# B&R Automation Studio project CombinedLinenSoiledA9KAN (part 16)

#### hlDFIICyclic.st - Cyclic code
```iecst
(********************************************************************
 * COPYRIGHT -- Microsoft
 ********************************************************************
 * Program: hlDFII
 * File: hlDFIICyclic.st
 * Author: hunholz
 * Created: April 05, 2011
 * Changed: November 14, 2011
 ********************************************************************
 * Implementation of program hlDFII
 ********************************************************************)

PROGRAM _CYCLIC

	// Init
	IF IFmnParam.Out.xParamOK AND NOT _xInitDone THEN

		brwcsconv(ADR(_sMNo), ADR(IFmnParam.Out.utfMachineNumber), 1);

		_xInitDone := TRUE;

	END_IF

	IF NOT _xReady AND IFmnEth.Out.xDataValid AND IFmnParam.Out.xParamOK AND HLDFII_RUN_CLIENT THEN

		//**********************
		// INITIALISIERUNG
		//***********************

		_sDBserv := USINT_TO_STRING(IFmnEth.Out.IP.bNetId1);
		_sDBserv := CONCAT(_sDBserv,'.');
		_sOkt := USINT_TO_STRING(IFmnEth.Out.IP.bNetId2);
		_sDBserv := CONCAT(_sDBserv,_sOkt);
		_sDBserv := CONCAT(_sDBserv,'.');
		_sOkt := USINT_TO_STRING(IFmnEth.Out.IP.bNetId3+hlDFIIPar.Mac.bDBservReg);
		_sDBserv := CONCAT(_sDBserv,_sOkt);
		_sDBserv := CONCAT(_sDBserv,'.');
		_sOkt := USINT_TO_STRING(hlDFIIPar.Mac.bDBservAdr);
		_sDBserv := CONCAT(_sDBserv,_sOkt);

		_sUdpHost := _sDBserv;

		brsstrcpy(ADR(_sInstance),ADR(hlDFIIPar.Mac.sServInst));

		IF hlDFIIPar.Mac.wDBservPort <> 0 THEN

			// Wenn der Port <> 0 ist, wird der SQL-Server direkt über den Port angesprochen

			_sDBserv := CONCAT(_sDBserv, ':');
			_sOkt 	 := UINT_TO_STRING(hlDFIIPar.Mac.wDBservPort);
			_sDBserv := CONCAT(_sDBserv, _sOkt);

		ELSE

			// Wenn mit der Instanz gearbeitet wird, muss auf dem PC der SQL-Browser-Dienst laufen

			IF LEN(_sInstance) > 0 THEN

				REPEAT

					_iFound := FIND(_sInstance,' ');

					IF _iFound <> 0 THEN
						_sInstance := DELETE(_sInstance,1,_iFound);
					END_IF

					UNTIL
					_iFound = 0 OR LEN(_sInstance) = 0
				END_REPEAT

				IF LEN(_sInstance) > 0 THEN
					_sDBserv := CONCAT(_sDBserv, '\');
					_sDBserv := CONCAT(_sDBserv, _sInstance);
				END_IF

			END_IF

		END_IF

		_xReady := TRUE;

		// UDP-Log vorbereiten

		_UdpOpen.enable	 := TRUE;
		_UdpOpen.pIfAddr := 0;
		_UdpOpen.port	 := HLDFII_UDP_PORT_LOG4NET;
		_UdpOpen.options := udpOPT_BROADCAST;

	ELSIF _xReady THEN

		//***********************************
		// ZYKLISCHE ABARBEITUNG
		//***********************************

		hlDFIIStat.wStatus := 0;

		//*********************************************************************************
		// Request scheduler
		//*********************************************************************************

		IF _eCmdStep = eCMD_SQLREQ_IDLE THEN

			CASE _wCmdCnt OF

				0:
					// Uhrzeit holen
					IF _bEventGetTime = 1 THEN
						// Auftrag starten
						_eCmdStep := eCMD_SQLREQ_WRITE_GETTIME;
						_bEventGetTime := 2;
					END_IF
				1:
					// Maschine registrieren
					IF _bEventRegMach = 1 AND brwcscmp(ADR(IFmnParam.Out.utfMachineNumber),ADR(MNPARAM_INVALID_MACHINENO)) <> 0 THEN
						// Auftrag starten
						_eCmdStep := eCMD_SQLREQ_WRITE_REGMACH;
						_bEventRegMach := 2;
					END_IF

				2:
					IF _xWaitReqProgByCatIsZero THEN

						IF IFhlDFII.In.ReqProgByCat.wRequest = 0 THEN

							_xWaitReqProgByCatIsZero := FALSE;
							IFhlDFII.Out.RespProgByCat.wResponse := 0;

						END_IF

					ELSE

						// Prüfen ob eine Programmnummer gelesen werden soll
						IF IFhlDFII.In.ReqProgByCat.wRequest = 1 OR IFhlDFII.In.ReqProgByCat.wRequest = 2 THEN

							IF IFhlDFII.Out.xConnected THEN

								_xWaitReqProgByCatIsZero := TRUE;
								// Auftrag starten
								_eCmdStep := eCMD_SQLREQ_GET_PROG_BY_CAT;
								IFhlDFII.Out.RespProgByCat.wResponse := ERR_FUB_BUSY;

							ELSE

								_xWaitReqProgByCatIsZero := TRUE;
								IFhlDFII.Out.RespProgByCat.wResponse := HLDFII_STAT_NO_CONNECTION;

							END_IF

						END_IF

					END_IF

				3:
					IF _xWaitReqMsgEvtIsZero THEN

						IF IFhlDFII.In.ReqMsgEvt.wRequest = 0 THEN
							_xWaitReqMsgEvtIsZero := FALSE;
							IFhlDFII.Out.RespMsgEvt.wResponse := 0;
						END_IF

					ELSE

						IF IFhlDFII.Out.xConnected THEN

							// Prüfen ob Meldungsevents geschrieben werden sollen
							IF IFhlDFII.In.ReqMsgEvt.wRequest = 1 THEN

								_xWaitReqMsgEvtIsZero := TRUE;

								IF IFhlDFII.In.ReqMsgEvt.bCntLines > 0 THEN
									_eCmdStep := eCMD_SQLREQ_WRITE_MSG;
									IFhlDFII.Out.RespMsgEvt.wResponse := ERR_FUB_BUSY;
								ELSE
									IFhlDFII.Out.RespMsgEvt.wResponse := IFhlDFII.In.ReqMsgEvt.wRequest;
								END_IF

							END_IF

						ELSE

							_xWaitReqMsgEvtIsZero := TRUE;
							IFhlDFII.Out.RespMsgEvt.wResponse := HLDFII_STAT_NO_CONNECTION;

						END_IF

					END_IF

				4:
					IF _xWaitReqCntBatchIsZero THEN

						IF IFhlDFII.In.ReqCntBatchEvt.wRequest = 0 THEN

							_xWaitReqCntBatchIsZero := FALSE;
							IFhlDFII.Out.RespCntBatchEvt.wResponse := 0;

						END_IF

					ELSE

						IF IFhlDFII.Out.xConnected THEN

							// Prüfen ob Zähler-Posten-Events geschrieben werden sollen
							IF IFhlDFII.In.ReqCntBatchEvt.wRequest = 1 THEN

								_xWaitReqCntBatchIsZero := TRUE;

								IF IFhlDFII.In.ReqCntBatchEvt.bCntLines > 0 THEN
									_eCmdStep := eCMD_SQLREQ_WRITE_CNTBATCHEVT;
									IFhlDFII.Out.RespCntBatchEvt.wResponse := ERR_FUB_BUSY;
								ELSE
									IFhlDFII.Out.RespCntBatchEvt.wResponse  := IFhlDFII.In.ReqCntBatchEvt.wRequest;
								END_IF
							END_IF

						ELSE

							_xWaitReqCntBatchIsZero := TRUE;
							IFhlDFII.Out.RespCntBatchEvt.wResponse := HLDFII_STAT_NO_CONNECTION;

						END_IF

					END_IF
				5:
					IF _xWaitReqCntCntIsZero THEN

						IF IFhlDFII.In.ReqCntCntEvt.wRequest = 0 THEN

							_xWaitReqCntCntIsZero := FALSE;
							IFhlDFII.Out.RespCntCntEvt.wResponse := 0;

						END_IF

					ELSE

						IF IFhlDFII.Out.xConnected THEN

							// Prüfen ob Zähler-Zähler-Events geschrieben werden sollen
							IF IFhlDFII.In.ReqCntCntEvt.wRequest = 1 THEN

								_xWaitReqCntCntIsZero := TRUE;

								IF IFhlDFII.In.ReqCntCntEvt.bCntLines > 0 THEN
									_eCmdStep := eCMD_SQLREQ_WRITE_CNTCNTEVT;
									IFhlDFII.Out.RespCntCntEvt.wResponse := ERR_FUB_BUSY;
								ELSE
									IFhlDFII.Out.RespCntCntEvt.wResponse  := IFhlDFII.In.ReqCntCntEvt.wRequest;
								END_IF
							END_IF

						ELSE

							_xWaitReqCntCntIsZero := TRUE;
							IFhlDFII.Out.RespCntCntEvt.wResponse := HLDFII_STAT_NO_CONNECTION;

						END_IF

					END_IF
				6:
					IF _xWaitReqCntTimIsZero THEN

						IF IFhlDFII.In.ReqCntTimEvt.wRequest = 0 THEN

							_xWaitReqCntTimIsZero := FALSE;
							IFhlDFII.Out.RespCntTimEvt.wResponse := 0;

						END_IF

					ELSE

						IF IFhlDFII.Out.xConnected THEN

							// Prüfen ob Zähler-Zeit-Events geschrieben werden sollen
							IF IFhlDFII.In.ReqCntTimEvt.wRequest = 1 THEN

								_xWaitReqCntTimIsZero := TRUE;

								IF IFhlDFII.In.ReqCntTimEvt.bCntLines > 0 THEN
									_eCmdStep := eCMD_SQLREQ_WRITE_CNTTIMEVT;
									IFhlDFII.Out.RespCntTimEvt.wResponse := ERR_FUB_BUSY;
								ELSE
									IFhlDFII.Out.RespCntTimEvt.wResponse  := IFhlDFII.In.ReqCntTimEvt.wRequest;
								END_IF
							END_IF

						ELSE

							_xWaitReqCntTimIsZero := TRUE;
							IFhlDFII.Out.RespCntTimEvt.wResponse := HLDFII_STAT_NO_CONNECTION;

						END_IF

					END_IF
				7:
					IF _xWaitReqCntDosIsZero THEN

						IF IFhlDFII.In.ReqCntDosEvt.wRequest = 0 THEN

							_xWaitReqCntDosIsZero := FALSE;
							IFhlDFII.Out.RespCntDosEvt.wResponse := 0;

						END_IF

					ELSE

						IF IFhlDFII.Out.xConnected THEN

							// Prüfen ob Zähler-Dosier-Events geschrieben werden sollen
							IF IFhlDFII.In.ReqCntDosEvt.wRequest = 1 THEN

								_xWaitReqCntDosIsZero := TRUE;

								IF IFhlDFII.In.ReqCntDosEvt.bCntLines > 0 THEN
									_eCmdStep := eCMD_SQLREQ_WRITE_CNTDOSEVT;
									IFhlDFII.Out.RespCntDosEvt.wResponse := ERR_FUB_BUSY;
								ELSE
									IFhlDFII.Out.RespCntDosEvt.wResponse  := IFhlDFII.In.ReqCntDosEvt.wRequest;
								END_IF

							END_IF

						ELSE

							_xWaitReqCntDosIsZero := TRUE;
							IFhlDFII.Out.RespCntDosEvt.wResponse := HLDFII_STAT_NO_CONNECTION;

						END_IF

					END_IF

			END_CASE

		END_IF

		//*********************************************************************************
		// Aufträge ausführen
		//*********************************************************************************

		CASE _eCmdStep OF

			eCMD_SQLREQ_IDLE:

				IF TRUE THEN

					IF _bEventGetTime <> 3 THEN
						_wCmdCnt := 0;
					ELSIF _bEventRegMach <> 3 THEN
						_wCmdCnt := 1;
					ELSE
						_wHelpCmdCnt := (_wHelpCmdCnt + 1) MOD 6;
						_wCmdCnt := _wHelpCmdCnt + 2;
					END_IF

				ELSE

					_xReady := FALSE;

				END_IF

			//*****************************************************
			// Auftrag: Programm nach Kategorie auslesen
			//*****************************************************
			eCMD_SQLREQ_GET_PROG_BY_CAT:

				IF _eStep = eSQLREQ_STEP_WAITFORCOMMAND THEN
					IFhlDFII.Out.RespProgByCat.bProgramNo 		:= 0;
					IFhlDFII.Out.RespProgByCat.sProgramName 	:= '';
					IFhlDFII.Out.RespProgByCat.rSoilfactor 		:= 1.0;
					IFhlDFII.Out.RespProgByCat.wLoadrate 		:= 100;
					IFhlDFII.Out.RespProgByCat.wColorIdxFor 	:= 0;
					IFhlDFII.Out.RespProgByCat.wColorIdxBack 	:= 15;
					_eStep := eSQLREQ_STEP_GPBC;
					_eCmdStep := eCMD_SQLREQ_GET_PROG_BY_CAT_w;

				ELSIF _eStep = eSQLREQ_STEP_ERROR THEN

					IFhlDFII.Out.RespProgByCat.wResponse := HLDFII_MSG_PROGBYCAT_ERR;
					_eCmdStep := eCMD_SQLREQ_IDLE;

				END_IF

			eCMD_SQLREQ_GET_PROG_BY_CAT_w:

				IF _eStep = eSQLREQ_STEP_WAITFORCOMMAND THEN
					IFhlDFII.Out.RespProgByCat.wResponse := IFhlDFII.In.ReqProgByCat.wRequest;
					_eCmdStep := eCMD_SQLREQ_IDLE;
				ELSIF _eStep = eSQLREQ_STEP_ERROR THEN
					IFhlDFII.Out.RespProgByCat.wResponse := HLDFII_MSG_PROGBYCAT_ERR;
					_eCmdStep := eCMD_SQLREQ_IDLE;
				END_IF

			//*****************************************************
			// Meldungen schreiben
			//*****************************************************
			eCMD_SQLREQ_WRITE_MSG:

				IF _eStep = eSQLREQ_STEP_WAITFORCOMMAND THEN
					_bCntWrMsg := 1;
					_eStep := eSQLREQ_STEP_WRMSG;
					_eCmdStep := eCMD_SQLREQ_WRITE_MSG_w;
				ELSIF _eStep = eSQLREQ_STEP_ERROR THEN
					IFhlDFII.Out.RespMsgEvt.wResponse := HLDFII_MSG_MSGEVT_ERR;
					_eCmdStep := eCMD_SQLREQ_IDLE;
				END_IF

			eCMD_SQLREQ_WRITE_MSG_w:

				IF _eStep = eSQLREQ_STEP_WAITFORCOMMAND THEN
					IFhlDFII.Out.RespMsgEvt.wResponse := IFhlDFII.In.ReqMsgEvt.wRequest;
					_eCmdStep := eCMD_SQLREQ_IDLE;
				ELSIF _eStep = eSQLREQ_STEP_ERROR THEN
					IFhlDFII.Out.RespMsgEvt.wResponse := HLDFII_MSG_MSGEVT_ERR;
					_eCmdStep := eCMD_SQLREQ_IDLE;
				END_IF

			//*****************************************************
			// Posten-Zählevents schreiben
			//*****************************************************
			eCMD_SQLREQ_WRITE_CNTBATCHEVT:

				IF _eStep = eSQLREQ_STEP_WAITFORCOMMAND THEN
					_bCntWrCntBatchEvt := 1;
					_eStep := eSQLREQ_STEP_WRCNTBATCHEVT;
					_eCmdStep := eCMD_SQLREQ_WRITE_CNTBATCHEVT_w;
				ELSIF _eStep = eSQLREQ_STEP_ERROR THEN
					IFhlDFII.Out.RespCntBatchEvt.wResponse := HLDFII_MSG_CNTBATCHEVT_ERR;
					_eCmdStep := eCMD_SQLREQ_IDLE;
				END_IF

			eCMD_SQLREQ_WRITE_CNTBATCHEVT_w:

				IF _eStep = eSQLREQ_STEP_WAITFORCOMMAND THEN
					IFhlDFII.Out.RespCntBatchEvt.wResponse := IFhlDFII.In.ReqCntBatchEvt.wRequest;
					_eCmdStep := eCMD_SQLREQ_IDLE;
				ELSIF _eStep = eSQLREQ_STEP_ERROR THEN
					IFhlDFII.Out.RespCntBatchEvt.wResponse := HLDFII_MSG_CNTBATCHEVT_ERR;
					_eCmdStep := eCMD_SQLREQ_IDLE;
				END_IF

			//*****************************************************
			// Zählerevents schreiben
			//*****************************************************
			eCMD_SQLREQ_WRITE_CNTCNTEVT:

				IF _eStep = eSQLREQ_STEP_WAITFORCOMMAND THEN
					_bCntWrCntCntEvt := 1;
					_eStep := eSQLREQ_STEP_WRCNTCNTEVT;
					_eCmdStep := eCMD_SQLREQ_WRITE_CNTCNTEVT_w;
				ELSIF _eStep = eSQLREQ_STEP_ERROR THEN
					IFhlDFII.Out.RespCntCntEvt.wResponse := HLDFII_MSG_CNTCNTEVT_ERR;
					_eCmdStep := eCMD_SQLREQ_IDLE;
				END_IF

			eCMD_SQLREQ_WRITE_CNTCNTEVT_w:

				IF _eStep = eSQLREQ_STEP_WAITFORCOMMAND THEN
					IFhlDFII.Out.RespCntCntEvt.wResponse := IFhlDFII.In.ReqCntCntEvt.wRequest;
					_eCmdStep := eCMD_SQLREQ_IDLE;
				ELSIF _eStep = eSQLREQ_STEP_ERROR THEN
					IFhlDFII.Out.RespCntCntEvt.wResponse := HLDFII_MSG_CNTCNTEVT_ERR;
					_eCmdStep := eCMD_SQLREQ_IDLE;
				END_IF

			//*****************************************************
			// Zeitevents schreiben
			//*****************************************************
			eCMD_SQLREQ_WRITE_CNTTIMEVT:

				IF _eStep = eSQLREQ_STEP_WAITFORCOMMAND THEN
					_bCntWrCntTimeEvt := 1;
					_eStep := eSQLREQ_STEP_WRCNTTIMEVT;
					_eCmdStep := eCMD_SQLREQ_WRITE_CNTTIMEVT_w;
				ELSIF _eStep = eSQLREQ_STEP_ERROR THEN
					IFhlDFII.Out.RespCntTimEvt.wResponse := HLDFII_MSG_CNTTIMEVT_ERR;
					_eCmdStep := eCMD_SQLREQ_IDLE;
				END_IF

			eCMD_SQLREQ_WRITE_CNTTIMEVT_w:

				IF _eStep = eSQLREQ_STEP_WAITFORCOMMAND THEN
					IFhlDFII.Out.RespCntTimEvt.wResponse := IFhlDFII.In.ReqCntTimEvt.wRequest;
					_eCmdStep := eCMD_SQLREQ_IDLE;
				ELSIF _eStep = eSQLREQ_STEP_ERROR THEN
					IFhlDFII.Out.RespCntTimEvt.wResponse := HLDFII_MSG_CNTTIMEVT_ERR;
					_eCmdStep := eCMD_SQLREQ_IDLE;
				END_IF

			//*****************************************************
			// Dosierevents schreiben
			//*****************************************************
			eCMD_SQLREQ_WRITE_CNTDOSEVT:

				IF _eStep = eSQLREQ_STEP_WAITFORCOMMAND THEN
					_bCntWrCntDoseEvt := 1;
					_eStep := eSQLREQ_STEP_WRCNTDOSEVT;
					_eCmdStep := eCMD_SQLREQ_WRITE_CNTDOSEVT_W;
				ELSIF _eStep = eSQLREQ_STEP_ERROR THEN
					IFhlDFII.Out.RespCntDosEvt.wResponse := HLDFII_MSG_CNTDOSEVT_ERR;
					_eCmdStep := eCMD_SQLREQ_IDLE;
				END_IF

			eCMD_SQLREQ_WRITE_CNTDOSEVT_W:

				IF _eStep = eSQLREQ_STEP_WAITFORCOMMAND THEN
					IFhlDFII.Out.RespCntDosEvt.wResponse := IFhlDFII.In.ReqCntDosEvt.wRequest;
					_eCmdStep := eCMD_SQLREQ_IDLE;
				ELSIF _eStep = eSQLREQ_STEP_ERROR THEN
					IFhlDFII.Out.RespCntDosEvt.wResponse := HLDFII_MSG_CNTDOSEVT_ERR;
					_eCmdStep := eCMD_SQLREQ_IDLE;
				END_IF

			//*****************************************************
			// Maschine registrieren
			//*****************************************************
			eCMD_SQLREQ_WRITE_REGMACH:

				IF _eStep = eSQLREQ_STEP_WAITFORCOMMAND THEN
					_eStep := eSQLREQ_STEP_REGMACH;
					_eCmdStep := eCMD_SQLREQ_WRITE_REGMACH_w;
				ELSIF _eStep = eSQLREQ_STEP_ERROR THEN
					_bEventRegMach := 255;
					_eCmdStep := eCMD_SQLREQ_IDLE;
				END_IF

			eCMD_SQLREQ_WRITE_REGMACH_w:

				IF _eStep = eSQLREQ_STEP_WAITFORCOMMAND THEN
					_bEventRegMach := 3;
					_eCmdStep := eCMD_SQLREQ_IDLE;
				ELSIF _eStep = eSQLREQ_STEP_ERROR THEN
					_bEventRegMach := 255;
					_eCmdStep := eCMD_SQLREQ_IDLE;
				END_IF

			//*****************************************************
			// Uhrzeit vom DB-Server holen
			//*****************************************************
			eCMD_SQLREQ_WRITE_GETTIME:

				IF _eStep = eSQLREQ_STEP_WAITFORCOMMAND THEN
					_eStep := eSQLREQ_STEP_GETTIME;
					_eCmdStep := eCMD_SQLREQ_WRITE_GETTIME_w;
				ELSIF _eStep = eSQLREQ_STEP_ERROR THEN
					_bEventGetTime := 255;
					_eCmdStep := eCMD_SQLREQ_IDLE;
				END_IF

			eCMD_SQLREQ_WRITE_GETTIME_w:

				IF _eStep = eSQLREQ_STEP_WAITFORCOMMAND THEN
					_bEventGetTime := 3;
					_eCmdStep := eCMD_SQLREQ_IDLE;
				ELSIF _eStep = eSQLREQ_STEP_ERROR THEN
					_bEventGetTime := 255;
					_eCmdStep := eCMD_SQLREQ_IDLE;
				END_IF

		END_CASE

		//*********************************************************************************
		// Verbindung nach ablauf der Idletime abbauen, wenn keine Aktion ist
		//*********************************************************************************

		IF _eStep = eSQLREQ_STEP_ERROR THEN

			_eStep := eSQLREQ_STEP_DISCONNECT;

		ELSIF (_eCmdStep = eCMD_SQLREQ_IDLE) AND(_eStep = eSQLREQ_STEP_WAITFORCOMMAND) THEN

			_GTCurrent(enable := TRUE);

			IF _GTCurrent.DT1 > _GTlastAction.DT1 THEN

				IF DiffDT(_GTCurrent.DT1, _GTlastAction.DT1) > hlDFIIPar.Mac.wIdletimeDisconnect THEN

					// Idletime abgelaufen, Verbindung abbauen
					_eStep := eSQLREQ_STEP_DISCONNECT;

				END_IF

			END_IF

		ELSE

			_GTlastAction(enable := TRUE);

		END_IF

		//*********************************************************************************
		// Verbindung bei Bedarf aufbauen
		//*********************************************************************************

		IF _eCmdStep <> eCMD_SQLREQ_IDLE AND _eStep = eSQLREQ_STEP_STOP THEN

			_eStep := eSQLREQ_STEP_CONNECT;

		END_IF

		//*********************************************************************************
		// SQL-Befehle ausführen
		//*********************************************************************************

		CASE _eStep OF

			eSQLREQ_STEP_STOP:

			eSQLREQ_STEP_WAITFORCOMMAND:

			(* Verbinde Datenbank *)
			eSQLREQ_STEP_CONNECT:

				_DFII_Connect.enable := TRUE;
				_DFII_Connect.databaseSystem := DB_SYSTEM_MS_SQL;
				_DFII_Connect.pUserName := ADR('plc');
				_DFII_Connect.pPassword := ADR('plc');
				_DFII_Connect.pServerName := ADR(_sDBserv);
				_DFII_Connect.pDatabaseName := ADR(hlDFIIPar.Mac.sDBname);
				_eStep := eSQLREQ_STEP_CONNECT_r;

			(* Warte bis mit Datenbank verbunden *)
			eSQLREQ_STEP_CONNECT_r:

				_DFII_Connect();

				IF _DFII_Connect.status = ERR_OK THEN

					// Verbindung Erfolgreich

					IF _DFII_Connect.connectionIdent = 0 THEN

						// Wenn Verbindung nicht möglich, immer erst wieder Zeit holen und Maschine registrieren
						_bEventRegMach := 1;
						_bEventGetTime := 1;
						IFhlDFII.Out.xConnected := FALSE;

						// Fehler ist Clientseitig
						_sLogEntryI := 'Client Fault: Connect failed! ';
						_sLogEntryI := CONCAT(_sLogEntryI,_sDBserv);
						_eStep := eSQLREQ_STEP_LOGRB_ERROR;

					ELSE

						IFhlDFII.Out.xConnected := TRUE;

						_sLogEntryI := WSTRING_TO_STRING(IFmnParam.Out.utfMachineNumber);
						_sLogEntryI := CONCAT(_sLogEntryI, '-hlDFII$tSUCC$tCONNECT');
						_InsertRB(wPtrWrite := _wPtrRBwrite, wPtrRead := _wPtrRBread, wPtrStart := _wPtrRBstart);

						_lConnectionIdent := _DFII_Connect.connectionIdent;
						_eStep := eSQLREQ_STEP_WAITFORCOMMAND;
					END_IF

				ELSIF _DFII_Connect.status <> ERR_FUB_BUSY THEN

					// Wenn Verbindung nicht möglich, immer erst wieder Zeit holen und Maschine registrieren
					_bEventRegMach := 1;
					_bEventGetTime := 1;
					IFhlDFII.Out.xConnected := FALSE;

					// Verbindung fehlerbehaftet
					IF _DFII_Connect.connectionIdent <> 0 THEN

						// Fehler ist Serverseitig, Fehlermeldung holen

						_lConnectionIdent := _DFII_Connect.connectionIdent;
						_sAction := 'Connect failed:';
						_eStep := eSQLREQ_STEP_GET_ERROR;

					ELSE

						// Keine Verbindung zustande gekommen
						_sLogEntryI := 'Connect failed! ';
						_sLogEntryI := CONCAT(_sLogEntryI,_sDBserv);

						_eStep := eSQLREQ_STEP_LOGRB_ERROR;

					END_IF

				END_IF

			(* Baue Datenbankverbindung ab *)
			eSQLREQ_STEP_DISCONNECT:

				IF _lConnectionIdent <> 0 THEN
					_DFII_Disconnect.enable := TRUE;
					_DFII_Disconnect.connectionIdent := _lConnectionIdent;
					_eStep := eSQLREQ_STEP_DISCONNECT_r;
				ELSE
					_eStep := eSQLREQ_STEP_STOP;
				END_IF

			(* Warte bis Verbindung abgebaut ist *)
			eSQLREQ_STEP_DISCONNECT_r:

				_DFII_Disconnect();

				IF _DFII_Disconnect.status <> ERR_FUB_BUSY THEN

					// Verbindung erfolgreich unterbrochen

					_sLogEntryI := WSTRING_TO_STRING(IFmnParam.Out.utfMachineNumber);
					_sLogEntryI := CONCAT(_sLogEntryI, '-hlDFII$tSUCC$tDISCONNECT');
					_InsertRB(wPtrWrite := _wPtrRBwrite, wPtrRead := _wPtrRBread, wPtrStart := _wPtrRBstart);

					_eStep := eSQLREQ_STEP_STOP;
					_lConnectionIdent := 0;

				END_IF

			(* Lese Programmnummer aus Datenbank *)
			eSQLREQ_STEP_GPBC:

				_sCat := IFhlDFII.In.ReqProgByCat.sCategoryNo_In;

				brsstrcpy(ADR(_sSQLstring), ADR('SELECT [ProgramNo], [ProgramName], [CategoryName], [LoadFactor], [SoiledFactor], [fgColorIndex], [bgColorIndex]  FROM [dbo].[vwCatToProg01] WHERE [MachineID] = N$''));
				brsstrcat(ADR(_sSQLstring), ADR(_sMNo));
				IF (IFhlDFII.In.ReqProgByCat.wRequest = 2) THEN
					brsstrcat(ADR(_sSQLstring),ADR('$' AND  LTRIM(RTRIM(CategoryNoAlpha)) =  LTRIM(RTRIM($''));
				ELSE
					brsstrcat(ADR(_sSQLstring),ADR('$' AND [CategoryNo] = '));
				END_IF
				brsstrcat(ADR(_sSQLstring),ADR(_sCat));
				IF (IFhlDFII.In.ReqProgByCat.wRequest = 2) THEN
					brsstrcat(ADR(_sSQLstring),ADR('$'))'));
				END_IF

				_DFII_DBExecute.enable := TRUE;
				_DFII_DBExecute.pSqlStatement := ADR(_sSQLstring);
				_DFII_DBExecute.connectionIdent := _lConnectionIdent;

				_eStep := eSQLREQ_STEP_GPBC_r;

			eSQLREQ_STEP_GPBC_r:

				_DFII_DBExecute();

				IF _DFII_DBExecute.status = ERR_OK THEN

					_eStep := eSQLREQ_STEP_GPBC_FETCH;

				ELSIF _DFII_DBExecute.status <> ERR_FUB_BUSY THEN

					IF _DFII_DBExecute.dbError = DB_SQL_NO_DATA THEN

						_eStep := eSQLREQ_STEP_WAITFORCOMMAND;

					ELSE

						_sAction := 'Get Program failed:';
						_eStep := eSQLREQ_STEP_GET_ERROR;

					END_IF

				END_IF

			(* Zeile holen *)
			eSQLREQ_STEP_GPBC_FETCH:

				_DFII_DBFetch.enable := TRUE;
				_DFII_DBFetch.connectionIdent := _lConnectionIdent;
				_eStep := eSQLREQ_STEP_GPBC_FETCH_r;

			eSQLREQ_STEP_GPBC_FETCH_r:

				_DFII_DBFetch();

				IF _DFII_DBFetch.status = ERR_OK THEN

					_bCol := 1;
					_eStep := eSQLREQ_STEP_GPBC_GETVAL;

				ELSIF _DFII_DBFetch.status <> ERR_FUB_BUSY THEN

					IF _DFII_DBFetch.dbError = DB_SQL_NO_DATA THEN

						_eStep := eSQLREQ_STEP_WAITFORCOMMAND;

					ELSE

						_sAction := 'Get Program failed (FETCH):';
						_eStep := eSQLREQ_STEP_GET_ERROR;

					END_IF

				END_IF

			(* Werte holen *)

			eSQLREQ_STEP_GPBC_GETVAL:

				_DFII_GetData.enable := TRUE;
				_DFII_GetData.connectionIdent := _lConnectionIdent;
				_DFII_GetData.columnIdx := _bCol;

				CASE _bCol OF

					1:	_DFII_GetData.pData := ADR(_iProgNo);
						_DFII_GetData.dataSize := SIZEOF(_iProgNo);
						_DFII_GetData.dataType := DB_SQL_SMALLINT;

					2: 	_DFII_GetData.pData := ADR(IFhlDFII.Out.RespProgByCat.sProgramName);
						_DFII_GetData.dataSize := SIZEOF(IFhlDFII.Out.RespProgByCat.sProgramName);
						_DFII_GetData.dataType := DB_SQL_CHAR;

					3: 	_DFII_GetData.pData := ADR(IFhlDFII.Out.RespProgByCat.sCategoryName);
						_DFII_GetData.dataSize := SIZEOF(IFhlDFII.Out.RespProgByCat.sCategoryName);
						_DFII_GetData.dataType := DB_SQL_CHAR;

					4: 	_DFII_GetData.pData := ADR(_rLoadfactor);
						_DFII_GetData.dataSize := SIZEOF(_rLoadfactor);
						_DFII_GetData.dataType := DB_SQL_REAL;

					5: 	_DFII_GetData.pData := ADR(IFhlDFII.Out.RespProgByCat.rSoilfactor);
						_DFII_GetData.dataSize := SIZEOF(IFhlDFII.Out.RespProgByCat.rSoilfactor);
						_DFII_GetData.dataType := DB_SQL_REAL;

					6: 	_DFII_GetData.pData := ADR(_diColIdxFor);
						_DFII_GetData.dataSize := SIZEOF(_diColIdxFor);
						_DFII_GetData.dataType := DB_SQL_INTEGER;

					7: 	_DFII_GetData.pData := ADR(_diColIdxBack);
						_DFII_GetData.dataSize := SIZEOF(_diColIdxBack);
						_DFII_GetData.dataType := DB_SQL_INTEGER;

				END_CASE

				_eStep := eSQLREQ_STEP_GPBC_GETVAL_r;

			eSQLREQ_STEP_GPBC_GETVAL_r:

				_DFII_GetData();

				IF _DFII_GetData.status = ERR_OK THEN

					_bCol := _bCol + 1;

					IF _bCol <= 7 THEN
						_eStep := eSQLREQ_STEP_GPBC_GETVAL;
					ELSE
						IF _iProgNo >= 0 AND _iProgNo <= 99 THEN

							IFhlDFII.Out.RespProgByCat.bProgramNo := INT_TO_USINT(_iProgNo);
							IFhlDFII.Out.RespProgByCat.wLoadrate := REAL_TO_UINT(_rLoadfactor);
							IFhlDFII.Out.RespProgByCat.wColorIdxFor := DINT_TO_UINT(_diColIdxFor);
							IFhlDFII.Out.RespProgByCat.wColorIdxBack := DINT_TO_UINT(_diColIdxBack);

						ELSE

							IFhlDFII.Out.RespProgByCat.bProgramNo := 0;
							IFhlDFII.Out.RespProgByCat.wLoadrate := 100;
							IFhlDFII.Out.RespProgByCat.wColorIdxFor := 0;
							IFhlDFII.Out.RespProgByCat.wColorIdxBack := 15;

						END_IF

						_sLogEntryI := WSTRING_TO_STRING(IFmnParam.Out.utfMachineNumber);
						_sLogEntryI := CONCAT(_sLogEntryI, '-hlDFII$tSUCC$tGET PROG BY CAT');
						_InsertRB(wPtrWrite := _wPtrRBwrite, wPtrRead := _wPtrRBread, wPtrStart := _wPtrRBstart);

						_eStep := eSQLREQ_STEP_WAITFORCOMMAND;

					END_IF

				ELSIF _DFII_GetData.status <> ERR_FUB_BUSY THEN
					_sAction := 'Get Program failed (VAL):';
					_eStep := eSQLREQ_STEP_GET_ERROR;
				END_IF

			// Meldungen per Prozedur schreiben
			eSQLREQ_STEP_WRMSG:

				IF _bCntWrMsg > IFhlDFII.In.ReqMsgEvt.bCntLines THEN

					_eStep := eSQLREQ_STEP_WAITFORCOMMAND;

				ELSE

					brsstrcpy(ADR(_sSQLstring), ADR('EXEC [dbo].[spInsMsgEvt01]  @MachineID = N$''));
					brsstrcat(ADR(_sSQLstring), ADR(_sMNo));
					brsstrcat(ADR(_sSQLstring), ADR('$''));

					brsstrcat(ADR(_sSQLstring),ADR(', @FunctionID = '));
					brsitoa(IFhlDFII.In.ReqMsgEvt.MsgHistList[_bCntWrMsg].wFunction_ID,ADR(_sFunctionID));
					brsstrcat(ADR(_sSQLstring),ADR(_sFunctionID));

					brsstrcat(ADR(_sSQLstring),ADR(', @MsgNo = '));
					brsitoa(IFhlDFII.In.ReqMsgEvt.MsgHistList[_bCntWrMsg].wMsgNumber,ADR(_sMsgNo));
					brsstrcat(ADR(_sSQLstring),ADR(_sMsgNo));

					brsstrcat(ADR(_sSQLstring),ADR(', @Instance = '));
					brsitoa(IFhlDFII.In.ReqMsgEvt.MsgHistList[_bCntWrMsg].wInstance,ADR(_sInstance));
					brsstrcat(ADR(_sSQLstring),ADR(_sInstance));

					brsstrcat(ADR(_sSQLstring),ADR(', @MsgClass = '));
					brsitoa(IFhlDFII.In.ReqMsgEvt.MsgHistList[_bCntWrMsg].wMsgClass,ADR(_sClass));
					brsstrcat(ADR(_sSQLstring),ADR(_sClass));

					brsstrcat(ADR(_sSQLstring),ADR(', @Event = '));
					brsitoa(IFhlDFII.In.ReqMsgEvt.MsgHistList[_bCntWrMsg].wEvent,ADR(_sEvent));
					brsstrcat(ADR(_sSQLstring),ADR(_sEvent));

					brsstrcat(ADR(_sSQLstring),ADR(', @TimeStamp = '));
					brsitoa(DT_TO_DINT(IFhlDFII.In.ReqMsgEvt.MsgHistList[_bCntWrMsg].TimeStampEvent),ADR(_sTimeStamp));
					brsstrcat(ADR(_sSQLstring),ADR(_sTimeStamp));

					brsstrcat(ADR(_sSQLstring),ADR(', @Time = '));
					brsitoa(IFhlDFII.In.ReqMsgEvt.MsgHistList[_bCntWrMsg].lTime,ADR(_sTime));
					brsstrcat(ADR(_sSQLstring),ADR(_sTime));

					// ##AH20111118
					brsstrcat(ADR(_sSQLstring),ADR(', @Attr1 = $''));
					brsstrcat(ADR(_sSQLstring),ADR(IFhlDFII.In.ReqMsgEvt.MsgHistList[_bCntWrMsg].sAttrTxt));

					brsstrcat(ADR(_sSQLstring),ADR('$', @Attr2 = '));
					brsitoa(IFhlDFII.In.ReqMsgEvt.MsgHistList[_bCntWrMsg].diAttr1,ADR(_sValue));
					brsstrcat(ADR(_sSQLstring),ADR(_sValue));

					brsstrcat(ADR(_sSQLstring),ADR(', @Attr3 = '));
					brsitoa(IFhlDFII.In.ReqMsgEvt.MsgHistList[_bCntWrMsg].diAttr2,ADR(_sValue));
					brsstrcat(ADR(_sSQLstring),ADR(_sValue));

					_DFII_DBExecute.enable := TRUE;
					_DFII_DBExecute.pSqlStatement := ADR(_sSQLstring);
					_DFII_DBExecute.connectionIdent := _lConnectionIdent;

					 _eStep := eSQLREQ_STEP_WRMSG_r;

				END_IF

			eSQLREQ_STEP_WRMSG_r:

				_DFII_DBExecute();

				IF _DFII_DBExecute.status = ERR_OK  OR _DFII_DBExecute.dbError = DB_SQL_NO_DATA THEN

					_sLogEntryI := WSTRING_TO_STRING(IFmnParam.Out.utfMachineNumber);
					_sLogEntryI := CONCAT(_sLogEntryI, '-hlDFII$tSUCC$tWRITE MESSAGE');
					_InsertRB(wPtrWrite := _wPtrRBwrite, wPtrRead := _wPtrRBread, wPtrStart := _wPtrRBstart);

					_bCntWrMsg := _bCntWrMsg + 1;
					_eStep := eSQLREQ_STEP_WRMSG;

				ELSIF _DFII_DBExecute.status <> ERR_FUB_BUSY THEN

					_sAction := 'Write Msg failed:';

					_eStep := eSQLREQ_STEP_GET_ERROR;

				END_IF

			// Postendaten schreiben
			eSQLREQ_STEP_WRCNTBATCHEVT:

				IF _bCntWrCntBatchEvt > IFhlDFII.In.ReqCntBatchEvt.bCntLines THEN

					 _eStep := eSQLREQ_STEP_WAITFORCOMMAND;

				ELSE

					CASE IFhlDFII.In.ReqCntBatchEvt.CntBatchEvtList[_bCntWrCntBatchEvt].bEvent OF

						MNCNT_BATCHEVENT_LOAD, MNCNT_BATCHEVENT_UNLOAD:

							_sSQLstring := 'EXEC [dbo].[spInsEventStat] ';

							_kgUSINT16toGUID(usintarray := IFhlDFII.In.ReqCntBatchEvt.CntBatchEvtList[_bCntWrCntBatchEvt].Batch.bBatchNo);

							IF IFhlDFII.In.ReqCntBatchEvt.CntBatchEvtList[_bCntWrCntBatchEvt].Batch.bTypeBatchNo = 0 THEN

								brsstrcat(ADR(_sSQLstring), ADR('@BatchID_INT = '));
								kgitoa_udint(num := kgBatchNoToUDINT(_kgUSINT16toGUID.GUID),str := _sUDINT);
								brsstrcat(ADR(_sSQLstring), ADR(_sUDINT));

							ELSE

								brsstrcat(ADR(_sSQLstring), ADR('@BatchID_GUID = $''));
								_kgGUIDtoSTRING(GUID := _kgUSINT16toGUID.GUID);
								brsstrcat(ADR(_sSQLstring), ADR(_kgGUIDtoSTRING.sOut));
								brsstrcat(ADR(_sSQLstring), ADR('$''));

							END_IF

							brsstrcat(ADR(_sSQLstring), ADR(', @MachineID = N$''));
							brsstrcat(ADR(_sSQLstring), ADR(_sMNo));
							brsstrcat(ADR(_sSQLstring), ADR('$''));

							brsstrcat(ADR(_sSQLstring), ADR(', @CategoryNoAlpha = $''));
							brsstrcat(ADR(_sSQLstring), ADR(IFhlDFII.In.ReqCntBatchEvt.CntBatchEvtList[_bCntWrCntBatchEvt].Batch.sCategory));
							brsstrcat(ADR(_sSQLstring), ADR('$''));

							brsstrcat(ADR(_sSQLstring), ADR(', @ProgNo = '));
							itoa(IFhlDFII.In.ReqCntBatchEvt.CntBatchEvtList[_bCntWrCntBatchEvt].bProgram, ADR(_sValue));
							brsstrcat(ADR(_sSQLstring), ADR(_sValue));

							brsstrcat(ADR(_sSQLstring), ADR(', @Selection = N$''));
							brwcsconv(ADR(_sMark), ADR(IFhlDFII.In.ReqCntBatchEvt.CntBatchEvtList[_bCntWrCntBatchEvt].Batch.utfMark), 1);
							brsstrcat(ADR(_sSQLstring), ADR(_sMark));
							brsstrcat(ADR(_sSQLstring), ADR('$''));

							brsstrcat(ADR(_sSQLstring), ADR(', @Time = $''));
							_mnParam_datetimetoa(dtTimestamp := IFhlDFII.In.ReqCntBatchEvt.CntBatchEvtList[_bCntWrCntBatchEvt].Batch.dtTimeStamp);
							brsstrcat(ADR(_sSQLstring), ADR(_mnParam_datetimetoa.sDateTime));
							brsstrcat(ADR(_sSQLstring), ADR('$'$R$L'));

							IF IFhlDFII.In.ReqCntBatchEvt.CntBatchEvtList[_bCntWrCntBatchEvt].Batch.bCntCustomers > 0 AND IFhlDFII.In.ReqCntBatchEvt.CntBatchEvtList[_bCntWrCntBatchEvt].Batch.bCntCustomers <= 8 THEN

								FOR _ii := 1 TO IFhlDFII.In.ReqCntBatchEvt.CntBatchEvtList[_bCntWrCntBatchEvt].Batch.bCntCustomers DO

									_idxCustomer := _ii - 1;

									brsstrcat(ADR(_sSQLstring), ADR('EXEC [dbo].[spInsEventStatItem_PartBatch] '));

									_kgUSINT16toGUID(usintarray := IFhlDFII.In.ReqCntBatchEvt.CntBatchEvtList[_bCntWrCntBatchEvt].Batch.bBatchNo);

									IF IFhlDFII.In.ReqCntBatchEvt.CntBatchEvtList[_bCntWrCntBatchEvt].Batch.bTypeBatchNo = 0 THEN

										brsstrcat(ADR(_sSQLstring), ADR('@BatchID_INT = '));
										kgitoa_udint(num := kgBatchNoToUDINT(_kgUSINT16toGUID.GUID),str := _sUDINT);
										brsstrcat(ADR(_sSQLstring), ADR(_sUDINT));

									ELSE

										brsstrcat(ADR(_sSQLstring), ADR('@BatchID_GUID = $''));
										_kgGUIDtoSTRING(GUID := _kgUSINT16toGUID.GUID);
										brsstrcat(ADR(_sSQLstring), ADR(_kgGUIDtoSTRING.sOut));
										brsstrcat(ADR(_sSQLstring), ADR('$''));

									END_IF

									brsstrcat(ADR(_sSQLstring), ADR(', @Machine = N$''));
									brsstrcat(ADR(_sSQLstring), ADR(_sMNo));
									brsstrcat(ADR(_sSQLstring), ADR('$''));

									brsstrcat(ADR(_sSQLstring), ADR(', @PartBatchID = '));
									brsitoa(_ii, ADR(_sValue));
									brsstrcat(ADR(_sSQLstring), ADR(_sValue));

									brsstrcat(ADR(_sSQLstring), ADR(', @ActualAmount = '));
									_sValue := REAL_TO_STRING(UINT_TO_REAL(IFhlDFII.In.ReqCntBatchEvt.CntBatchEvtList[_bCntWrCntBatchEvt].Batch.PartBatch[_idxCustomer].wCustomWeight)/10.0);
									brsstrcat(ADR(_sSQLstring), ADR(_sValue));

									brsstrcat(ADR(_sSQLstring), ADR(', @Customer = $''));
									brsstrcat(ADR(_sSQLstring), ADR(IFhlDFII.In.ReqCntBatchEvt.CntBatchEvtList[_bCntWrCntBatchEvt].Batch.PartBatch[_idxCustomer].sCustomNo));
									brsstrcat(ADR(_sSQLstring), ADR('$''));

									IF IFhlDFII.In.ReqCntBatchEvt.CntBatchEvtList[_bCntWrCntBatchEvt].bEvent = MNCNT_BATCHEVENT_LOAD THEN

										brsstrcat(ADR(_sSQLstring), ADR(', @FromOutside = 1, @ToOutside = 0 '));

									END_IF

									IF IFhlDFII.In.ReqCntBatchEvt.CntBatchEvtList[_bCntWrCntBatchEvt].bEvent = MNCNT_BATCHEVENT_UNLOAD THEN

										brsstrcat(ADR(_sSQLstring), ADR(', @FromOutside = 0, @ToOutside = 1  '));

									END_IF

									brsstrcat(ADR(_sSQLstring), ADR(', @FromName = N$''));
									brsstrcat(ADR(_sSQLstring), ADR(IFhlDFII.In.ReqCntBatchEvt.CntBatchEvtList[_bCntWrCntBatchEvt].FromLocation.sNameId));
									brsstrcat(ADR(_sSQLstring), ADR('$''));

									brsstrcat(ADR(_sSQLstring), ADR(', @ToName = N$''));
									brsstrcat(ADR(_sSQLstring), ADR(IFhlDFII.In.ReqCntBatchEvt.CntBatchEvtList[_bCntWrCntBatchEvt].ToLocation.sNameId));
									brsstrcat(ADR(_sSQLstring), ADR('$''));

									brsstrcat(ADR(_sSQLstring), ADR(', @Time = $''));
									_mnParam_datetimetoa(dtTimestamp := IFhlDFII.In.ReqCntBatchEvt.CntBatchEvtList[_bCntWrCntBatchEvt].Batch.dtTimeStamp);
									brsstrcat(ADR(_sSQLstring), ADR(_mnParam_datetimetoa.sDateTime));
									brsstrcat(ADR(_sSQLstring), ADR('$'$R$L'));

								END_FOR

								_DFII_DBExecute.enable := TRUE;
								_DFII_DBExecute.pSqlStatement := ADR(_sSQLstring);
								_DFII_DBExecute.connectionIdent := _lConnectionIdent;

							END_IF

							_sSQLBatchEventString := _sSQLstring;

							_eStep := eSQLREQ_STEP_WRCNTBATCHEVT_r;

						MNCNT_BATCHEVENT_CHANGEDATA:

							_sSQLstring := 'EXEC [dbo].[spUpdEventStat] ';

							_kgUSINT16toGUID(usintarray := IFhlDFII.In.ReqCntBatchEvt.CntBatchEvtList[_bCntWrCntBatchEvt].Batch.bBatchNo);

							IF IFhlDFII.In.ReqCntBatchEvt.CntBatchEvtList[_bCntWrCntBatchEvt].Batch.bTypeBatchNo = 0 THEN

								brsstrcat(ADR(_sSQLstring), ADR('@BatchID_INT = '));
								kgitoa_udint(num := kgBatchNoToUDINT(_kgUSINT16toGUID.GUID),str := _sUDINT);
								brsstrcat(ADR(_sSQLstring), ADR(_sUDINT));

							ELSE

								brsstrcat(ADR(_sSQLstring), ADR('@BatchID_GUID = $''));
								_kgGUIDtoSTRING(GUID := _kgUSINT16toGUID.GUID);
								brsstrcat(ADR(_sSQLstring), ADR(_kgGUIDtoSTRING.sOut));
								brsstrcat(ADR(_sSQLstring), ADR('$''));

							END_IF

							brsstrcat(ADR(_sSQLstring), ADR(', @MachineID = N$''));
							brsstrcat(ADR(_sSQLstring), ADR(_sMNo));
							brsstrcat(ADR(_sSQLstring), ADR('$''));

							brsstrcat(ADR(_sSQLstring), ADR(', @CategoryNoAlpha = $''));
							brsstrcat(ADR(_sSQLstring), ADR(IFhlDFII.In.ReqCntBatchEvt.CntBatchEvtList[_bCntWrCntBatchEvt].Batch.sCategory));
							brsstrcat(ADR(_sSQLstring), ADR('$''));

							brsstrcat(ADR(_sSQLstring), ADR(', @ProgNo = '));
							itoa(IFhlDFII.In.ReqCntBatchEvt.CntBatchEvtList[_bCntWrCntBatchEvt].bProgram, ADR(_sValue));
							brsstrcat(ADR(_sSQLstring), ADR(_sValue));

							brsstrcat(ADR(_sSQLstring), ADR(', @Selection = N$''));
							brwcsconv(ADR(_sMark), ADR(IFhlDFII.In.ReqCntBatchEvt.CntBatchEvtList[_bCntWrCntBatchEvt].Batch.utfMark), 1);
							brsstrcat(ADR(_sSQLstring), ADR(_sMark));
							brsstrcat(ADR(_sSQLstring), ADR('$''));

							brsstrcat(ADR(_sSQLstring), ADR(', @Time = $''));
							_mnParam_datetimetoa(dtTimestamp := IFhlDFII.In.ReqCntBatchEvt.CntBatchEvtList[_bCntWrCntBatchEvt].Batch.dtTimeStamp);
							brsstrcat(ADR(_sSQLstring), ADR(_mnParam_datetimetoa.sDateTime));
							brsstrcat(ADR(_sSQLstring), ADR('$'$R$L'));

							IF IFhlDFII.In.ReqCntBatchEvt.CntBatchEvtList[_bCntWrCntBatchEvt].Batch.bCntCustomers > 0 AND IFhlDFII.In.ReqCntBatchEvt.CntBatchEvtList[_bCntWrCntBatchEvt].Batch.bCntCustomers <= 8 THEN

								FOR _ii := 1 TO IFhlDFII.In.ReqCntBatchEvt.CntBatchEvtList[_bCntWrCntBatchEvt].Batch.bCntCustomers DO

									_idxCustomer := _ii - 1;

									brsstrcat(ADR(_sSQLstring), ADR('EXEC [dbo].[spUpdEventStatItem_PartBatch] '));

									_kgUSINT16toGUID(usintarray := IFhlDFII.In.ReqCntBatchEvt.CntBatchEvtList[_bCntWrCntBatchEvt].Batch.bBatchNo);

									IF IFhlDFII.In.ReqCntBatchEvt.CntBatchEvtList[_bCntWrCntBatchEvt].Batch.bTypeBatchNo = 0 THEN

										brsstrcat(ADR(_sSQLstring), ADR('@BatchID_INT = '));
										kgitoa_udint(num := kgBatchNoToUDINT(_kgUSINT16toGUID.GUID),str := _sUDINT);
										brsstrcat(ADR(_sSQLstring), ADR(_sUDINT));

									ELSE

										brsstrcat(ADR(_sSQLstring), ADR('@BatchID_GUID = $''));
										_kgGUIDtoSTRING(GUID := _kgUSINT16toGUID.GUID);
										brsstrcat(ADR(_sSQLstring), ADR(_kgGUIDtoSTRING.sOut));
										brsstrcat(ADR(_sSQLstring), ADR('$''));

									END_IF

									brsstrcat(ADR(_sSQLstring), ADR(', @Machine = N$''));
									brsstrcat(ADR(_sSQLstring), ADR(_sMNo));
									brsstrcat(ADR(_sSQLstring), ADR('$''));

									brsstrcat(ADR(_sSQLstring), ADR(', @PartBatchID = '));
									brsitoa(_ii, ADR(_sValue));
									brsstrcat(ADR(_sSQLstring), ADR(_sValue));

									brsstrcat(ADR(_sSQLstring), ADR(', @ActualAmount = '));
									_sValue := REAL_TO_STRING(UINT_TO_REAL(IFhlDFII.In.ReqCntBatchEvt.CntBatchEvtList[_bCntWrCntBatchEvt].Batch.PartBatch[_idxCustomer].wCustomWeight)/10.0);
									brsstrcat(ADR(_sSQLstring), ADR(_sValue));

									brsstrcat(ADR(_sSQLstring), ADR(', @Customer = $''));
									brsstrcat(ADR(_sSQLstring), ADR(IFhlDFII.In.ReqCntBatchEvt.CntBatchEvtList[_bCntWrCntBatchEvt].Batch.PartBatch[_idxCustomer].sCustomNo));
									brsstrcat(ADR(_sSQLstring), ADR('$''));

									brsstrcat(ADR(_sSQLstring), ADR(', @Time = $''));
									_mnParam_datetimetoa(dtTimestamp := IFhlDFII.In.ReqCntBatchEvt.CntBatchEvtList[_bCntWrCntBatchEvt].Batch.dtTimeStamp);
									brsstrcat(ADR(_sSQLstring), ADR(_mnParam_datetimetoa.sDateTime));
									brsstrcat(ADR(_sSQLstring), ADR('$'$R$L'));

								END_FOR

								_DFII_DBExecute.enable := TRUE;
								_DFII_DBExecute.pSqlStatement := ADR(_sSQLstring);
								_DFII_DBExecute.connectionIdent := _lConnectionIdent;

							END_IF

							_sSQLBatchEventString := _sSQLstring;

							_eStep := eSQLREQ_STEP_WRCNTBATCHEVT_r;

						MNCNT_BATCHEVENT_DELETE:

							_bCntWrCntBatchEvt := _bCntWrCntBatchEvt + 1;

					END_CASE

				END_IF

			eSQLREQ_STEP_WRCNTBATCHEVT_r:

				_DFII_DBExecute();

				IF _DFII_DBExecute.status = ERR_OK  OR _DFII_DBExecute.dbError = DB_SQL_NO_DATA THEN

					_sLogEntryI := WSTRING_TO_STRING(IFmnParam.Out.utfMachineNumber);
					_sLogEntryI := CONCAT(_sLogEntryI, '-hlDFII$tSUCC$tWRITE BATCH EVENT');
					_InsertRB(wPtrWrite := _wPtrRBwrite, wPtrRead := _wPtrRBread, wPtrStart := _wPtrRBstart);

					_bCntWrCntBatchEvt := _bCntWrCntBatchEvt + 1;
					_eStep := eSQLREQ_STEP_WRCNTBATCHEVT;

				ELSIF _DFII_DBExecute.status <> ERR_FUB_BUSY THEN

					_sAction := 'Write Batch failed:';
					_eStep := eSQLREQ_STEP_GET_ERROR;

				END_IF

			eSQLREQ_STEP_WRCNTCNTEVT:

				IF _bCntWrCntCntEvt > IFhlDFII.In.ReqCntCntEvt.bCntLines THEN

					_eStep := eSQLREQ_STEP_WAITFORCOMMAND;

				ELSE

					CASE IFhlDFII.In.ReqCntCntEvt.CntCounterEvtList[_bCntWrCntCntEvt].bType OF

						MNCNT_COUNTERTYPE_WATER:

							_sSQLstring := 'EXEC [dbo].[spInsEventStatItem_Water] ';

							brsstrcat(ADR(_sSQLstring), ADR('@Machine = N$''));
							brsstrcat(ADR(_sSQLstring), ADR(_sMNo));
							brsstrcat(ADR(_sSQLstring), ADR('$''));

							_kgUSINT16toGUID(usintarray := IFhlDFII.In.ReqCntCntEvt.CntCounterEvtList[_bCntWrCntCntEvt].BatchNo);

							IF NOT kgGUIDisZero(_kgUSINT16toGUID.GUID) THEN

								IF IFhlDFII.In.ReqCntCntEvt.CntCounterEvtList[_bCntWrCntCntEvt].bTypeBatchNo = 0 THEN

									brsstrcat(ADR(_sSQLstring), ADR(', @BatchID_INT = '));
									kgitoa_udint(num := kgBatchNoToUDINT(_kgUSINT16toGUID.GUID),str := _sUDINT);
									brsstrcat(ADR(_sSQLstring), ADR(_sUDINT));

								ELSE

									brsstrcat(ADR(_sSQLstring), ADR(', @BatchID_GUID = $''));
									_kgGUIDtoSTRING(GUID := _kgUSINT16toGUID.GUID);
									brsstrcat(ADR(_sSQLstring), ADR(_kgGUIDtoSTRING.sOut));
									brsstrcat(ADR(_sSQLstring), ADR('$''));

								END_IF

							END_IF

							brsstrcat(ADR(_sSQLstring), ADR(', @ActualAmount = '));
							_sValue := REAL_TO_STRING(UDINT_TO_REAL(IFhlDFII.In.ReqCntCntEvt.CntCounterEvtList[_bCntWrCntCntEvt].lAmount));
							brsstrcat(ADR(_sSQLstring), ADR(_sValue));

							brsstrcat(ADR(_sSQLstring), ADR(', @TargetAmount = '));
							_sValue := REAL_TO_STRING(UDINT_TO_REAL(IFhlDFII.In.ReqCntCntEvt.CntCounterEvtList[_bCntWrCntCntEvt].lNomAmount));
							brsstrcat(ADR(_sSQLstring), ADR(_sValue));

//							IF IFhlDFII.In.ReqCntCntEvt.CntCounterEvtList[_bCntWrCntCntEvt].Source.bCompartment > 0 THEN
//
//								brsstrcat(ADR(_sSQLstring), ADR(', @FromChamber = '));
//								_sValue := USINT_TO_STRING(IFhlDFII.In.ReqCntCntEvt.CntCounterEvtList[_bCntWrCntCntEvt].Source.bCompartment);
//								brsstrcat(ADR(_sSQLstring), ADR(_sValue));
//
//							ELSE

								brsstrcat(ADR(_sSQLstring), ADR(', @FromName = N$''));
								brsstrcat(ADR(_sSQLstring), ADR(IFhlDFII.In.ReqCntCntEvt.CntCounterEvtList[_bCntWrCntCntEvt].Source.sNameId));
								brsstrcat(ADR(_sSQLstring), ADR('$''));

//							END_IF

							IF IFhlDFII.In.ReqCntCntEvt.CntCounterEvtList[_bCntWrCntCntEvt].Source.bLocationExt > 0 THEN

								brsstrcat(ADR(_sSQLstring), ADR(', @FromOutside = 1'));

							ELSE

								brsstrcat(ADR(_sSQLstring), ADR(', @FromOutside = 0'));

							END_IF

//							IF IFhlDFII.In.ReqCntCntEvt.CntCounterEvtList[_bCntWrCntCntEvt].Destination.bCompartment > 0 THEN
//
//								brsstrcat(ADR(_sSQLstring), ADR(', @ToChamber = '));
//								_sValue := USINT_TO_STRING(IFhlDFII.In.ReqCntCntEvt.CntCounterEvtList[_bCntWrCntCntEvt].Destination.bCompartment);
//								brsstrcat(ADR(_sSQLstring), ADR(_sValue));
//
//							ELSE

								brsstrcat(ADR(_sSQLstring), ADR(', @ToName = N$''));
								brsstrcat(ADR(_sSQLstring), ADR(IFhlDFII.In.ReqCntCntEvt.CntCounterEvtList[_bCntWrCntCntEvt].Destination.sNameId));
								brsstrcat(ADR(_sSQLstring), ADR('$''));

//							END_IF

							IF IFhlDFII.In.ReqCntCntEvt.CntCounterEvtList[_bCntWrCntCntEvt].Destination.bLocationExt > 0 THEN

								brsstrcat(ADR(_sSQLstring), ADR(', @ToOutside = 1'));

							ELSE

								brsstrcat(ADR(_sSQLstring), ADR(', @ToOutside = 0'));

							END_IF

							brsstrcat(ADR(_sSQLstring), ADR(', @Time = $''));
							_mnParam_datetimetoa(dtTimestamp := IFhlDFII.In.ReqCntCntEvt.CntCounterEvtList[_bCntWrCntCntEvt].dtTimeStamp);
							brsstrcat(ADR(_sSQLstring), ADR(_mnParam_datetimetoa.sDateTime));
							brsstrcat(ADR(_sSQLstring), ADR('$''));

							_DFII_DBExecute.enable := TRUE;
							_DFII_DBExecute.pSqlStatement := ADR(_sSQLstring);
							_DFII_DBExecute.connectionIdent := _lConnectionIdent;

							_eStep := eSQLREQ_STEP_WRCNTCNTEVT_r;

						MNCNT_COUNTERTYPE_TEMPERATURE:

							_sSQLstring := 'EXEC [dbo].[spInsEventStatItem_Temperature] ';

							brsstrcat(ADR(_sSQLstring), ADR('@Machine = N$''));
							brsstrcat(ADR(_sSQLstring), ADR(_sMNo));
							brsstrcat(ADR(_sSQLstring), ADR('$''));

							_kgUSINT16toGUID(usintarray := IFhlDFII.In.ReqCntCntEvt.CntCounterEvtList[_bCntWrCntCntEvt].BatchNo);

							IF NOT kgGUIDisZero(_kgUSINT16toGUID.GUID) THEN

								IF IFhlDFII.In.ReqCntCntEvt.CntCounterEvtList[_bCntWrCntCntEvt].bTypeBatchNo = 0 THEN

									brsstrcat(ADR(_sSQLstring), ADR(', @BatchID_INT = '));
									kgitoa_udint(num := kgBatchNoToUDINT(_kgUSINT16toGUID.GUID),str := _sUDINT);
									brsstrcat(ADR(_sSQLstring), ADR(_sUDINT));

								ELSE

									brsstrcat(ADR(_sSQLstring), ADR(', @BatchID_GUID = $''));
									_kgGUIDtoSTRING(GUID := _kgUSINT16toGUID.GUID);
									brsstrcat(ADR(_sSQLstring), ADR(_kgGUIDtoSTRING.sOut));
									brsstrcat(ADR(_sSQLstring), ADR('$''));

								END_IF

							END_IF

							brsstrcat(ADR(_sSQLstring), ADR(', @ActualAmount = '));
							_sValue := REAL_TO_STRING(UDINT_TO_REAL(IFhlDFII.In.ReqCntCntEvt.CntCounterEvtList[_bCntWrCntCntEvt].lAmount));
							brsstrcat(ADR(_sSQLstring), ADR(_sValue));

							brsstrcat(ADR(_sSQLstring), ADR(', @TargetAmount = '));
							_sValue := REAL_TO_STRING(UDINT_TO_REAL(IFhlDFII.In.ReqCntCntEvt.CntCounterEvtList[_bCntWrCntCntEvt].lNomAmount));
							brsstrcat(ADR(_sSQLstring), ADR(_sValue));

//							IF IFhlDFII.In.ReqCntCntEvt.CntCounterEvtList[_bCntWrCntCntEvt].Destination.bCompartment > 0 THEN
//
//								brsstrcat(ADR(_sSQLstring), ADR(', @LocationChamber = '));
//								_sValue := USINT_TO_STRING(IFhlDFII.In.ReqCntCntEvt.CntCounterEvtList[_bCntWrCntCntEvt].Destination.bCompartment);
//								brsstrcat(ADR(_sSQLstring), ADR(_sValue));
//
//							ELSE

								brsstrcat(ADR(_sSQLstring), ADR(', @LocationName = N$''));
								brsstrcat(ADR(_sSQLstring), ADR(IFhlDFII.In.ReqCntCntEvt.CntCounterEvtList[_bCntWrCntCntEvt].Destination.sNameId));
								brsstrcat(ADR(_sSQLstring), ADR('$''));

//							END_IF

							IF IFhlDFII.In.ReqCntCntEvt.CntCounterEvtList[_bCntWrCntCntEvt].Destination.bLocationExt > 0 THEN

								brsstrcat(ADR(_sSQLstring), ADR(', @LocationOutside = 1'));

							ELSE

								brsstrcat(ADR(_sSQLstring), ADR(', @LocationOutside = 0'));

							END_IF

							brsstrcat(ADR(_sSQLstring), ADR(', @Time = $''));
							_mnParam_datetimetoa(dtTimestamp := IFhlDFII.In.ReqCntCntEvt.CntCounterEvtList[_bCntWrCntCntEvt].dtTimeStamp);
							brsstrcat(ADR(_sSQLstring), ADR(_mnParam_datetimetoa.sDateTime));
							brsstrcat(ADR(_sSQLstring), ADR('$''));

							_DFII_DBExecute.enable := TRUE;
							_DFII_DBExecute.pSqlStatement := ADR(_sSQLstring);
							_DFII_DBExecute.connectionIdent := _lConnectionIdent;

							_eStep := eSQLREQ_STEP_WRCNTCNTEVT_r;

						MNCNT_COUNTERTYPE_STEAM, MNCNT_COUNTERTYPE_ELECTRICENERGY, MNCNT_COUNTERTYPE_GAS:

							IF IFhlDFII.In.ReqCntCntEvt.CntCounterEvtList[_bCntWrCntCntEvt].bType = MNCNT_COUNTERTYPE_STEAM THEN
								_sSQLstring := 'EXEC [dbo].[spInsEventStatItem_Steam] ';
							ELSIF IFhlDFII.In.ReqCntCntEvt.CntCounterEvtList[_bCntWrCntCntEvt].bType = MNCNT_COUNTERTYPE_GAS THEN
								_sSQLstring := 'EXEC [dbo].[spInsEventStatItem_Gas] ';
							ELSE
								_sSQLstring := 'EXEC [dbo].[spInsEventStatItem_Energy] ';
							END_IF

							brsstrcat(ADR(_sSQLstring), ADR('@Machine = N$''));
							brsstrcat(ADR(_sSQLstring), ADR(_sMNo));
							brsstrcat(ADR(_sSQLstring), ADR('$''));

							_kgUSINT16toGUID(usintarray := IFhlDFII.In.ReqCntCntEvt.CntCounterEvtList[_bCntWrCntCntEvt].BatchNo);

							IF NOT kgGUIDisZero(_kgUSINT16toGUID.GUID) THEN

								IF IFhlDFII.In.ReqCntCntEvt.CntCounterEvtList[_bCntWrCntCntEvt].bTypeBatchNo = 0 THEN

									brsstrcat(ADR(_sSQLstring), ADR(', @BatchID_INT = '));
									kgitoa_udint(num := kgBatchNoToUDINT(_kgUSINT16toGUID.GUID),str := _sUDINT);
									brsstrcat(ADR(_sSQLstring), ADR(_sUDINT));

								ELSE

									brsstrcat(ADR(_sSQLstring), ADR(', @BatchID_GUID = $''));
									_kgGUIDtoSTRING(GUID := _kgUSINT16toGUID.GUID);
									brsstrcat(ADR(_sSQLstring), ADR(_kgGUIDtoSTRING.sOut));
									brsstrcat(ADR(_sSQLstring), ADR('$''));

								END_IF

							END_IF

							brsstrcat(ADR(_sSQLstring), ADR(', @ActualAmount = '));
							_sValue := REAL_TO_STRING(UDINT_TO_REAL(IFhlDFII.In.ReqCntCntEvt.CntCounterEvtList[_bCntWrCntCntEvt].lAmount));
							brsstrcat(ADR(_sSQLstring), ADR(_sValue));

//							IF IFhlDFII.In.ReqCntCntEvt.CntCounterEvtList[_bCntWrCntCntEvt].Source.bCompartment > 0 THEN
//
//								brsstrcat(ADR(_sSQLstring), ADR(', @FromChamber = '));
//								_sValue := USINT_TO_STRING(IFhlDFII.In.ReqCntCntEvt.CntCounterEvtList[_bCntWrCntCntEvt].Source.bCompartment);
//								brsstrcat(ADR(_sSQLstring), ADR(_sValue));
//
//							ELSE

								brsstrcat(ADR(_sSQLstring), ADR(', @FromName = N$''));
								brsstrcat(ADR(_sSQLstring), ADR(IFhlDFII.In.ReqCntCntEvt.CntCounterEvtList[_bCntWrCntCntEvt].Source.sNameId));
								brsstrcat(ADR(_sSQLstring), ADR('$''));

//							END_IF

							IF IFhlDFII.In.ReqCntCntEvt.CntCounterEvtList[_bCntWrCntCntEvt].Source.bLocationExt > 0 THEN

								brsstrcat(ADR(_sSQLstring), ADR(', @FromOutside = 1'));

							ELSE

								brsstrcat(ADR(_sSQLstring), ADR(', @FromOutside = 0'));

							END_IF

//							IF IFhlDFII.In.ReqCntCntEvt.CntCounterEvtList[_bCntWrCntCntEvt].Destination.bCompartment > 0 THEN
//
//								brsstrcat(ADR(_sSQLstring), ADR(', @ToChamber = '));
//								_sValue := USINT_TO_STRING(IFhlDFII.In.ReqCntCntEvt.CntCounterEvtList[_bCntWrCntCntEvt].Destination.bCompartment);
//								brsstrcat(ADR(_sSQLstring), ADR(_sValue));
//
//							ELSE

								brsstrcat(ADR(_sSQLstring), ADR(', @ToName = N$''));
								brsstrcat(ADR(_sSQLstring), ADR(IFhlDFII.In.ReqCntCntEvt.CntCounterEvtList[_bCntWrCntCntEvt].Destination.sNameId));
								brsstrcat(ADR(_sSQLstring), ADR('$''));

//							END_IF

							IF IFhlDFII.In.ReqCntCntEvt.CntCounterEvtList[_bCntWrCntCntEvt].Destination.bLocationExt > 0 THEN

								brsstrcat(ADR(_sSQLstring), ADR(', @ToOutside = 1'));

							ELSE

								brsstrcat(ADR(_sSQLstring), ADR(', @ToOutside = 0'));

							END_IF

							brsstrcat(ADR(_sSQLstring), ADR(', @Time = $''));
							_mnParam_datetimetoa(dtTimestamp := IFhlDFII.In.ReqCntCntEvt.CntCounterEvtList[_bCntWrCntCntEvt].dtTimeStamp);
							brsstrcat(ADR(_sSQLstring), ADR(_mnParam_datetimetoa.sDateTime));
							brsstrcat(ADR(_sSQLstring), ADR('$''));

							_DFII_DBExecute.enable := TRUE;
							_DFII_DBExecute.pSqlStatement := ADR(_sSQLstring);
							_DFII_DBExecute.connectionIdent := _lConnectionIdent;

							_eStep := eSQLREQ_STEP_WRCNTCNTEVT_r;

						ELSE

							_bCntWrCntCntEvt := _bCntWrCntCntEvt + 1;

					END_CASE

				END_IF

			eSQLREQ_STEP_WRCNTCNTEVT_r:

				_DFII_DBExecute();

				IF _DFII_DBExecute.status = ERR_OK  OR _DFII_DBExecute.dbError = DB_SQL_NO_DATA THEN

					_sLogEntryI := WSTRING_TO_STRING(IFmnParam.Out.utfMachineNumber);
					_sLogEntryI := CONCAT(_sLogEntryI, '-hlDFII$tSUCC$tWRITE COUNT EVENT');
					_InsertRB(wPtrWrite := _wPtrRBwrite, wPtrRead := _wPtrRBread, wPtrStart := _wPtrRBstart);

					_bCntWrCntCntEvt := _bCntWrCntCntEvt + 1;
					_eStep := eSQLREQ_STEP_WRCNTCNTEVT;

				ELSIF _DFII_DBExecute.status <> ERR_FUB_BUSY THEN

					_sAction := 'Write Counter failed:';
					_eStep := eSQLREQ_STEP_GET_ERROR;

				END_IF

			// Zeitzähler senden

			eSQLREQ_STEP_WRCNTTIMEVT:

				IF _bCntWrCntTimeEvt > IFhlDFII.In.ReqCntTimEvt.bCntLines THEN

					_eStep := eSQLREQ_STEP_WAITFORCOMMAND;

				ELSE

					_sSQLstring := 'EXEC [dbo].[spInsEventStatItem_StateTime] ';

					brsstrcat(ADR(_sSQLstring), ADR('@Machine = N$''));
					brsstrcat(ADR(_sSQLstring), ADR(_sMNo));
					brsstrcat(ADR(_sSQLstring), ADR('$''));

					brsstrcat(ADR(_sSQLstring), ADR(', @ActualAmount = '));
					_sValue := REAL_TO_STRING(UDINT_TO_REAL(IFhlDFII.In.ReqCntTimEvt.CntTimerEvtList[_bCntWrCntTimeEvt].lAmount));
					brsstrcat(ADR(_sSQLstring), ADR(_sValue));

					IF IFhlDFII.In.ReqCntTimEvt.CntTimerEvtList[_bCntWrCntTimeEvt].bState = MNCNT_TIMERSTATE_PAUSED THEN

						brsstrcat(ADR(_sSQLstring), ADR(', @State = $'PAUSED$''));

						CASE IFhlDFII.In.ReqCntTimEvt.CntTimerEvtList[_bCntWrCntTimeEvt].bSubState OF

							MNCNT_TIMERSUBSTATE_OFF:

								brsstrcat(ADR(_sSQLstring), ADR(', @SubState = $'OFF$''));

							MNCNT_TIMERSUBSTATE_STOP:

								brsstrcat(ADR(_sSQLstring), ADR(', @SubState = $'STOP$''));

							MNCNT_TIMERSUBSTATE_INTFAULT:

								brsstrcat(ADR(_sSQLstring), ADR(', @SubState = $'INTFAULT$''));

							MNCNT_TIMERSUBSTATE_EXTFAULT:

								brsstrcat(ADR(_sSQLstring), ADR(', @SubState = $'EXTFAULT$''));

							MNCNT_TIMERSUBSTATE_SAFESTOP:

								brsstrcat(ADR(_sSQLstring), ADR(', @SubState = $'SAFESTOP$''));

							MNCNT_TIMERSUBSTATE_EMERGENCYSTP:

								brsstrcat(ADR(_sSQLstring), ADR(', @SubState = $'EMERGSTOP$''));

							ELSE

								brsstrcat(ADR(_sSQLstring), ADR(', @SubState = $'$''));

						END_CASE

					ELSIF IFhlDFII.In.ReqCntTimEvt.CntTimerEvtList[_bCntWrCntTimeEvt].bState = MNCNT_TIMERSTATE_WAIT THEN

						brsstrcat(ADR(_sSQLstring), ADR(', @State = $'WAIT$''));

						CASE IFhlDFII.In.ReqCntTimEvt.CntTimerEvtList[_bCntWrCntTimeEvt].bSubState OF

							MNCNT_TIMERSUBSTATE_LOADING:

								brsstrcat(ADR(_sSQLstring), ADR(', @SubState = $'LOADING$''));

							MNCNT_TIMERSUBSTATE_UNLOADING:

								brsstrcat(ADR(_sSQLstring), ADR(', @SubState = $'UNLOADING$''));

							MNCNT_TIMERSUBSTATE_DOSING:

								brsstrcat(ADR(_sSQLstring), ADR(', @SubState = $'DOSING$''));

							MNCNT_TIMERSUBSTATE_WATERLEVEL:

								brsstrcat(ADR(_sSQLstring), ADR(', @SubState = $'WATERLEVEL$''));

							MNCNT_TIMERSUBSTATE_TEMPERATURE:

								brsstrcat(ADR(_sSQLstring), ADR(', @SubState = $'TEMP$''));

							MNCNT_TIMERSUBSTATE_DISINFECTION:

								brsstrcat(ADR(_sSQLstring), ADR(', @SubState = $'DISINFECT$''));

							MNCNT_TIMERSUBSTATE_AIRPRESSURE:

								brsstrcat(ADR(_sSQLstring), ADR(', @SubState = $'AIRPRESS$''));

							ELSE

								brsstrcat(ADR(_sSQLstring), ADR(', @SubState = $'$''));

						END_CASE

					ELSIF IFhlDFII.In.ReqCntTimEvt.CntTimerEvtList[_bCntWrCntTimeEvt].bState = MNCNT_TIMERSTATE_ACTIVE THEN

						brsstrcat(ADR(_sSQLstring), ADR(', @State = $'ACTIVE$''));

						CASE IFhlDFII.In.ReqCntTimEvt.CntTimerEvtList[_bCntWrCntTimeEvt].bSubState OF

							MNCNT_TIMERSUBSTATE_WASHING:

								brsstrcat(ADR(_sSQLstring), ADR(', @SubState = $'WASHING$''));

							MNCNT_TIMERSUBSTATE_PREPERATION:

								brsstrcat(ADR(_sSQLstring), ADR(', @SubState = $'PREP$''));

							MNCNT_TIMERSUBSTATE_TRANSFER:

								brsstrcat(ADR(_sSQLstring), ADR(', @SubState = $'TRANSFER$''));

							MNCNT_TIMERSUBSTATE_PREPFORSTOP:

								brsstrcat(ADR(_sSQLstring), ADR(', @SubState = $'PREPFORSTOP$''));

							ELSE

								brsstrcat(ADR(_sSQLstring), ADR(', @SubState = $'$''));

						END_CASE

					ELSE

						brsstrcat(ADR(_sSQLstring), ADR(', @State = $'$', @SubState = $'$''));

					END_IF

					brsstrcat(ADR(_sSQLstring), ADR(', @Time = $''));
					_mnParam_datetimetoa(dtTimestamp := IFhlDFII.In.ReqCntTimEvt.CntTimerEvtList[_bCntWrCntTimeEvt].dtTimeStamp);
					brsstrcat(ADR(_sSQLstring), ADR(_mnParam_datetimetoa.sDateTime));
					brsstrcat(ADR(_sSQLstring), ADR('$''));

					_DFII_DBExecute.enable := TRUE;
					_DFII_DBExecute.pSqlStatement := ADR(_sSQLstring);
					_DFII_DBExecute.connectionIdent := _lConnectionIdent;

					_eStep := eSQLREQ_STEP_WRCNTTIMEVT_r;

				END_IF

			eSQLREQ_STEP_WRCNTTIMEVT_r:

				_DFII_DBExecute();

				IF _DFII_DBExecute.status = ERR_OK  OR _DFII_DBExecute.dbError = DB_SQL_NO_DATA THEN

					_sLogEntryI := WSTRING_TO_STRING(IFmnParam.Out.utfMachineNumber);
					_sLogEntryI := CONCAT(_sLogEntryI, '-hlDFII$tSUCC$tWRITE TIME EVENT');
					_InsertRB(wPtrWrite := _wPtrRBwrite, wPtrRead := _wPtrRBread, wPtrStart := _wPtrRBstart);

					_bCntWrCntTimeEvt := _bCntWrCntTimeEvt + 1;
					_eStep := eSQLREQ_STEP_WRCNTTIMEVT;

				ELSIF _DFII_DBExecute.status <> ERR_FUB_BUSY THEN

					_sAction := 'Write Time failed:';
					_eStep := eSQLREQ_STEP_GET_ERROR;

				END_IF

			// Dosierevents schreiben

			eSQLREQ_STEP_WRCNTDOSEVT:

				IF _bCntWrCntDoseEvt > IFhlDFII.In.ReqCntDosEvt.bCntLines THEN

					_eStep := eSQLREQ_STEP_WAITFORCOMMAND;

				ELSE

					_sSQLstring := 'EXEC [dbo].[spInsEventStatItem_Chemical] ';

					brsstrcat(ADR(_sSQLstring), ADR('@Machine = N$''));
					brsstrcat(ADR(_sSQLstring), ADR(_sMNo));
					brsstrcat(ADR(_sSQLstring), ADR('$''));

					_kgUSINT16toGUID(usintarray := IFhlDFII.In.ReqCntDosEvt.CntDosingEvtList[_bCntWrCntDoseEvt].DosingEvent.BatchNo);

					IF NOT kgGUIDisZero(_kgUSINT16toGUID.GUID) THEN

						IF IFhlDFII.In.ReqCntDosEvt.CntDosingEvtList[_bCntWrCntDoseEvt].DosingEvent.bTypeBatchNo = 0 THEN

							brsstrcat(ADR(_sSQLstring), ADR(', @BatchID_INT = '));
							kgitoa_udint(num := kgBatchNoToUDINT(_kgUSINT16toGUID.GUID),str := _sUDINT);
							brsstrcat(ADR(_sSQLstring), ADR(_sUDINT));

						ELSE

							brsstrcat(ADR(_sSQLstring), ADR(', @BatchID_GUID = $''));
							_kgGUIDtoSTRING(GUID := _kgUSINT16toGUID.GUID);
							brsstrcat(ADR(_sSQLstring), ADR(_kgGUIDtoSTRING.sOut));
							brsstrcat(ADR(_sSQLstring), ADR('$''));

						END_IF

					END_IF

					brsstrcat(ADR(_sSQLstring), ADR(', @ActualAmount = '));
					_sValue := REAL_TO_STRING(IFhlDFII.In.ReqCntDosEvt.CntDosingEvtList[_bCntWrCntDoseEvt].DosingEvent.rAmount);
					brsstrcat(ADR(_sSQLstring), ADR(_sValue));

					brsstrcat(ADR(_sSQLstring), ADR(', @TargetAmount = '));
					_sValue := REAL_TO_STRING(IFhlDFII.In.ReqCntDosEvt.CntDosingEvtList[_bCntWrCntDoseEvt].DosingEvent.rNomAmount);
					brsstrcat(ADR(_sSQLstring), ADR(_sValue));

					brsstrcat(ADR(_sSQLstring), ADR(', @Unit = $''));
					brsstrcat(ADR(_sSQLstring), ADR(IFhlDFII.In.ReqCntDosEvt.CntDosingEvtList[_bCntWrCntDoseEvt].DosingEvent.sUnit));
					brsstrcat(ADR(_sSQLstring), ADR('$''));

					_sDoseName := WSTRING_TO_STRING(IFhlDFII.In.ReqCntDosEvt.CntDosingEvtList[_bCntWrCntDoseEvt].DosingEvent.utfName);

					brsstrcat(ADR(_sSQLstring), ADR(', @Name = N$''));
					brsstrcat(ADR(_sSQLstring), ADR(_sDoseName));
					brsstrcat(ADR(_sSQLstring), ADR('$''));

					brsstrcat(ADR(_sSQLstring), ADR(', @FromName = N$''));
					brsstrcat(ADR(_sSQLstring), ADR(IFhlDFII.In.ReqCntDosEvt.CntDosingEvtList[_bCntWrCntDoseEvt].DosingEvent.Source.sNameId));
					brsstrcat(ADR(_sSQLstring), ADR('$''));

					IF IFhlDFII.In.ReqCntDosEvt.CntDosingEvtList[_bCntWrCntDoseEvt].DosingEvent.Source.bLocationExt > 0 THEN

						brsstrcat(ADR(_sSQLstring), ADR(', @FromOutside = 1'));

					ELSE

						brsstrcat(ADR(_sSQLstring), ADR(', @FromOutside = 0'));

					END_IF

					brsstrcat(ADR(_sSQLstring), ADR(', @ToName = N$''));
					brsstrcat(ADR(_sSQLstring), ADR(IFhlDFII.In.ReqCntDosEvt.CntDosingEvtList[_bCntWrCntDoseEvt].DosingEvent.Destination.sNameId));
					brsstrcat(ADR(_sSQLstring), ADR('$''));

					IF IFhlDFII.In.ReqCntDosEvt.CntDosingEvtList[_bCntWrCntDoseEvt].DosingEvent.Destination.bLocationExt > 0 THEN

						brsstrcat(ADR(_sSQLstring), ADR(', @ToOutside = 1'));

					ELSE

						brsstrcat(ADR(_sSQLstring), ADR(', @ToOutside = 0'));

					END_IF

					brsstrcat(ADR(_sSQLstring), ADR(', @Time = $''));
					_mnParam_datetimetoa(dtTimestamp := IFhlDFII.In.ReqCntDosEvt.CntDosingEvtList[_bCntWrCntDoseEvt].DosingEvent.dtTimeStamp);
					brsstrcat(ADR(_sSQLstring), ADR(_mnParam_datetimetoa.sDateTime));
					brsstrcat(ADR(_sSQLstring), ADR('$''));

					_DFII_DBExecute.enable := TRUE;
					_DFII_DBExecute.pSqlStatement := ADR(_sSQLstring);
					_DFII_DBExecute.connectionIdent := _lConnectionIdent;

					_eStep := eSQLREQ_STEP_WRCNTDOSEVT_r;

				END_IF

			eSQLREQ_STEP_WRCNTDOSEVT_r:

				_DFII_DBExecute();

				IF _DFII_DBExecute.status = ERR_OK  OR _DFII_DBExecute.dbError = DB_SQL_NO_DATA THEN

					_sLogEntryI := WSTRING_TO_STRING(IFmnParam.Out.utfMachineNumber);
					_sLogEntryI := CONCAT(_sLogEntryI, '-hlDFII$tSUCC$tWRITE DOSING EVENT');
					_InsertRB(wPtrWrite := _wPtrRBwrite, wPtrRead := _wPtrRBread, wPtrStart := _wPtrRBstart);

					_bCntWrCntDoseEvt := _bCntWrCntDoseEvt + 1;
					_eStep := eSQLREQ_STEP_WRCNTDOSEVT;

				ELSIF _DFII_DBExecute.status <> ERR_FUB_BUSY THEN

					_sAction := 'Write Dosing failed:';
					_eStep := eSQLREQ_STEP_GET_ERROR;

				END_IF

			// Maschine registrieren
			eSQLREQ_STEP_REGMACH:

				brsstrcpy(ADR(_sSQLstring), ADR('EXEC [dbo].[spRegMachine01]  @MachineID = N$''));
				brsstrcat(ADR(_sSQLstring), ADR(_sMNo));
				brsstrcat(ADR(_sSQLstring), ADR('$''));

				brsstrcat(ADR(_sSQLstring),ADR(', @ShortName = $''));
				brwcsconv(ADR(_sShortName),ADR(mnParamStatAd.HeaderVersion.utfMachineType),1);
				brsstrcat(ADR(_sSQLstring),ADR(_sShortName));
				brsstrcat(ADR(_sSQLstring),ADR('$''));

				brsstrcat(ADR(_sSQLstring),ADR(', @Name = $''));
				brwcsconv(ADR(_sName),ADR(mnParamStatAd.utfMachineName),1);
				brsstrcat(ADR(_sSQLstring),ADR(_sName));
				brsstrcat(ADR(_sSQLstring),ADR('$''));

				_DFII_DBExecute.enable := TRUE;
				_DFII_DBExecute.pSqlStatement := ADR(_sSQLstring);
				_DFII_DBExecute.connectionIdent := _lConnectionIdent;

				_eStep := eSQLREQ_STEP_REGMACH_r;

			eSQLREQ_STEP_REGMACH_r:

				_DFII_DBExecute();

				IF _DFII_DBExecute.status = ERR_OK  OR _DFII_DBExecute.dbError = DB_SQL_NO_DATA THEN

					_sLogEntryI := WSTRING_TO_STRING(IFmnParam.Out.utfMachineNumber);
					_sLogEntryI := CONCAT(_sLogEntryI, '-hlDFII$tSUCC$tREGMACHINE');
					_InsertRB(wPtrWrite := _wPtrRBwrite, wPtrRead := _wPtrRBread, wPtrStart := _wPtrRBstart);

					_eStep := eSQLREQ_STEP_WAITFORCOMMAND;

				ELSIF _DFII_DBExecute.status <> ERR_FUB_BUSY THEN

					_sAction := 'Reg. Machine failed:';
					_eStep := eSQLREQ_STEP_GET_ERROR;

				END_IF

			// Uhrzeit von DB lesen
			eSQLREQ_STEP_GETTIME:

				_sSQLstring := 'SELECT DATEDIFF(s,$'1970-01-01T00:00:00$',GETDATE())';

				_DFII_DBExecute.enable := TRUE;
				_DFII_DBExecute.pSqlStatement := ADR(_sSQLstring);
				_DFII_DBExecute.connectionIdent := _lConnectionIdent;

				_eStep := eSQLREQ_STEP_GETTIME_r;

			eSQLREQ_STEP_GETTIME_r:

				_DFII_DBExecute();

				IF _DFII_DBExecute.status = ERR_OK THEN

					_eStep := eSQLREQ_STEP_GETTIME_FETCH;

				ELSIF _DFII_DBExecute.status <> ERR_FUB_BUSY THEN

					_sAction := 'Get Time failed:';
					_eStep := eSQLREQ_STEP_GET_ERROR;

				END_IF

			(* Zeile holen *)
			eSQLREQ_STEP_GETTIME_FETCH:

				_DFII_DBFetch.enable := TRUE;
				_DFII_DBFetch.connectionIdent := _lConnectionIdent;
				_eStep := eSQLREQ_STEP_GETTIME_FETCH_r;

			eSQLREQ_STEP_GETTIME_FETCH_r:

				_DFII_DBFetch();

				IF _DFII_DBFetch.status = ERR_OK THEN

					_bCol := 1;
					_eStep := eSQLREQ_STEP_GETTIME_GETVAL;

				ELSIF _DFII_DBFetch.status <> ERR_FUB_BUSY THEN

					IF _DFII_DBFetch.dbError = DB_SQL_NO_DATA THEN

						_eStep := eSQLREQ_STEP_WAITFORCOMMAND;

					ELSE

						_sAction := 'Get Time failed (FETCH):';
						_eStep := eSQLREQ_STEP_GET_ERROR;

					END_IF

				END_IF

			(* Werte holen *)

			eSQLREQ_STEP_GETTIME_GETVAL:

				_DFII_GetData.enable := TRUE;
				_DFII_GetData.connectionIdent := _lConnectionIdent;
				_DFII_GetData.columnIdx := _bCol;

				_diTime := -1;
				_DFII_GetData.pData := ADR(_diTime);
				_DFII_GetData.dataSize := SIZEOF(_diTime);
				_DFII_GetData.dataType := DB_SQL_INTEGER;

				_eStep := eSQLREQ_STEP_GETTIME_GETVAL_r;

			eSQLREQ_STEP_GETTIME_GETVAL_r:

				_DFII_GetData();

				IF _DFII_GetData.status = ERR_OK THEN

					IF _diTime > 0 THEN

						_DTSetTime(enable := TRUE, DT1 := DINT_TO_DT(_diTime));

					END_IF

					_sLogEntryI := WSTRING_TO_STRING(IFmnParam.Out.utfMachineNumber);
					_sLogEntryI := CONCAT(_sLogEntryI, '-hlDFII$tSUCC$tGETTIME');
					_InsertRB(wPtrWrite := _wPtrRBwrite, wPtrRead := _wPtrRBread, wPtrStart := _wPtrRBstart);

					_eStep := eSQLREQ_STEP_WAITFORCOMMAND;

				ELSIF _DFII_GetData.status <> ERR_FUB_BUSY THEN
					_sAction := 'Get Time failed (VAL):';
					_eStep := eSQLREQ_STEP_GET_ERROR;
				END_IF

			(* Lese Fehler aus *)
			eSQLREQ_STEP_GET_ERROR:

				IF _lConnectionIdent = 0 THEN
					hlDFIIStat.sStatus := 'Connect failed !';
					_eStep := eSQLREQ_STEP_ERROR;
				ELSE
					brsmemset(ADR(hlDFIIStat.sStatus),0,SIZEOF(hlDFIIStat.sStatus));
					_DFII_DBErrMsg.enable := TRUE;
					_DFII_DBErrMsg.connectionIdent := _lConnectionIdent;
					_DFII_DBErrMsg.pErrorMessage := ADR(hlDFIIStat.sStatus);
					_DFII_DBErrMsg.errorMessageSize := SIZEOF(hlDFIIStat.sStatus);
					_eStep := eSQLREQ_STEP_GET_ERROR_r;
				END_IF

			(* Warte bis Fehler ausgelesen *)
			eSQLREQ_STEP_GET_ERROR_r:

				_DFII_DBErrMsg();

				IF _DFII_DBErrMsg.status = ERR_OK THEN

					_sLogEntryI := WSTRING_TO_STRING(IFmnParam.Out.utfMachineNumber);
					_sLogEntryI := CONCAT(_sLogEntryI, '-hlDFII$tWARN$t');
					_sLogEntryI := CONCAT(_sLogEntryI, _sAction);
					_sLogEntryI := CONCAT(_sLogEntryI, hlDFIIStat.sStatus);

					_eStep := eSQLREQ_STEP_LOGRB_ERROR;

				ELSIF _DFII_DBErrMsg.status <> ERR_FUB_BUSY THEN

					hlDFIIStat.sStatus := ' DBErrMsg.status = ';
					_sValue := UINT_TO_STRING(_DFII_DBErrMsg.status);
					hlDFIIStat.sStatus := CONCAT(hlDFIIStat.sStatus, _sValue);

					_sLogEntryI := WSTRING_TO_STRING(IFmnParam.Out.utfMachineNumber);
					_sLogEntryI := CONCAT(_sLogEntryI, '-hlDFII$tWARN$t');
					_sLogEntryI := CONCAT(_sLogEntryI, _sAction);
					_sLogEntryI := CONCAT(_sLogEntryI, hlDFIIStat.sStatus);

					_eStep := eSQLREQ_STEP_LOGRB_ERROR;

				END_IF

			eSQLREQ_STEP_LOGRB_ERROR:

				_InsertRB(wPtrWrite := _wPtrRBwrite, wPtrRead := _wPtrRBread, wPtrStart := _wPtrRBstart);
				_eStep := eSQLREQ_STEP_LOG_ERROR;

			eSQLREQ_STEP_LOG_ERROR:

				_kgArLogWrite.logLevel 	:= arlogLEVEL_WARNING;
				_kgArLogWrite.text		:= LEFT(_sLogEntryI, 127);
				_kgArLogWrite();

				IF _kgArLogWrite.status <> ERR_FUB_BUSY THEN
					brsmemset(ADR(_sLogEntryI), 0, SIZEOF(_sLogEntryI));
					_eStep := eSQLREQ_STEP_LOG_ERROR1;
				END_IF

			eSQLREQ_STEP_LOG_ERROR1:

				_kgArLogWrite.logLevel 	:= arlogLEVEL_WARNING;
				_kgArLogWrite.text		:= LEFT(_sSQLstring, 127);
				_kgArLogWrite();

				IF _kgArLogWrite.status <> ERR_FUB_BUSY THEN
					_eStep := eSQLREQ_STEP_ERROR;
				END_IF

			(* Fehlerschritt *)
			eSQLREQ_STEP_ERROR:

		END_CASE

		// Wenn Maschinenregistrierung fehlerhaft war, wiederholen nach ca. 1 Minute
		TONrepReg(IN := _bEventRegMach = 255, PT := T#60s);
		IF TONrepReg.Q THEN
			_bEventRegMach := 1;
		END_IF
		// Wenn Zeit lesen fehlerhaft war, wiederholen nach ca. 1 Minute
		TONrepGettime(IN := _bEventGetTime = 255, PT := T#60s);
		IF TONrepGettime.Q THEN
			_bEventGetTime := 1;
		END_IF

		// UDP Logging

		CASE _wStepUdp OF

			0:
				_UdpOpen();
				IF _UdpOpen.status = ERR_OK THEN
					_wStepUdp := 1;
				END_IF

			1:
				_ReadRB(wPtrWrite := _wPtrRBwrite, wPtrStart := _wPtrRBstart, wPtrRead := _wPtrRBread);

				IF _ReadRB.wStatus = ERR_OK THEN
					_wStepUdp := 2;
					_UdpSend.enable := TRUE;
					_UdpSend.ident := _UdpOpen.ident;
					_UdpSend.pHost := ADR(_sUdpHost);
					_UdpSend.port := HLDFII_UDP_PORT_LOG4NET;
					_UdpSend.pData := ADR(_sLogEntry);
					_UdpSend.datalen := SIZEOF(_sLogEntry);
				END_IF

			2:
				_UdpSend();
				IF _UdpSend.status <> ERR_FUB_BUSY THEN
					_wStepUdp := 1;
				END_IF

		END_CASE

		hlDFIIStat.wStatus := SEL(IFhlDFII.Out.xConnected,HLDFII_STAT_NO_CONNECTION, HLDFII_STAT_OK);
		IFhlDFII.Out.wStatus := SEL(IFhlDFII.Out.xConnected,HLDFII_STAT_NO_CONNECTION, HLDFII_STAT_OK);

	ELSE

		IF IFmnEth.Out.xDataValid AND IFmnParam.Out.xParamOK THEN

			hlDFIIStat.wStatus := HLDFII_STAT_DISABLED;
			IFhlDFII.Out.wStatus := HLDFII_STAT_DISABLED;

		ELSE

			hlDFIIStat.wStatus := HLDFII_STAT_INIT;
			IFhlDFII.Out.wStatus := HLDFII_STAT_INIT;

		END_IF

	END_IF

	// Debughilfe für _sSQLstring
	_wStartDebug := LIMIT(0,_wStartDebug, 992);
	_sDebugSQLstring ACCESS (ADR(_sSQLBatchEventString)+_wStartDebug);

END_PROGRAM
```

#### hlDFIIInit.st - Initialization code
```iecst
(********************************************************************
 * COPYRIGHT -- Microsoft
 ********************************************************************
 * Program: hlDFII
 * File: hlDFIIInit.st
 * Author: hunholz
 * Created: April 05, 2011
 ********************************************************************
 * Implementation of program hlDFII
 ********************************************************************)

PROGRAM _INIT

	// Packet-Version auslesen mit MO_ver aus SYS_lib und für den Additional Status zur Verfügung stellen

	_sPkgName := 'hlDFII';

	IF ( MO_ver(ADR(_sPkgName), 0, ADR(_VerStruc)) = 0 ) THEN

		brsmemcpy(ADR(hlDFIIStatAd.sPkgVersion), ADR(_VerStruc.version), SIZEOF(_VerStruc.version));

	ELSE

		hlDFIIStatAd.sPkgVersion := '---';

	END_IF

	// Init

	_xInitDone := FALSE;
	_xReady := FALSE;
	_eStep := eSQLREQ_STEP_STOP;
	_eCmdStep := eCMD_SQLREQ_IDLE;
	_bEventRegMach := 1;
	_bEventGetTime := 1;
	_lConnectionIdent := 0;
	_wCmdCnt := 0;
	_GTlastAction(enable := TRUE);
	brsmemset(ADR(hlDFIIStat),0,SIZEOF(hlDFIIStat));

	// Create Log
	//****************************************************************************************************************
	// Log erzeugen
	//****************************************************************************************************************

	_kgArLogWrite.enable := TRUE;
	_kgArLogWrite.ident := 0;
	_kgArLogWrite.errornr := 50010;

	_AsArLogCreate(enable := TRUE, pName := ADR('hlDFIIL'), len := 4096*4, memType := arlogUSRROM);

	IF _AsArLogCreate.status = ERR_OK THEN

		_kgArLogWrite.ident := _AsArLogCreate.ident;

	ELSIF _AsArLogCreate.status = arlogERR_EXISTING THEN

		_AsArLogGetInfo(enable := TRUE, pName := ADR('hlDFIIL'));

		IF _AsArLogGetInfo.status = ERR_OK THEN

			_kgArLogWrite.ident := _AsArLogGetInfo.ident;

		END_IF

	END_IF

	//****************************************************************************************************************
	// Ringbuffer for Logs
	//****************************************************************************************************************

	_kgRBcreateDFIIlog(sName := '_dfiilogrb', bMemType := doTEMP, wCntEntry := 10, lLenEntry := SIZEOF(_sLogEntry), wPtrWrite := _wPtrRBwrite, wPtrRead := _wPtrRBread, wPtrStart := _wPtrRBstart);

	IF _kgRBcreateDFIIlog.wStatus = ERR_OK THEN

		_wPtrRBloc := 0;

		_xRBReady := TRUE;

		_InsertRB.doIdent := _kgRBcreateDFIIlog.doIdent;
		_InsertRB.doLen := _kgRBcreateDFIIlog.doLen;
		_InsertRB.lLenEntry := SIZEOF(_sLogEntry);
		_InsertRB.pEntry := ADR(_sLogEntryI);

		_ReadRB.doIdent := _kgRBcreateDFIIlog.doIdent;
		_ReadRB.doLen := _kgRBcreateDFIIlog.doLen;
		_ReadRB.lLenEntry := SIZEOF(_sLogEntry);
		_ReadRB.pEntry := ADR(_sLogEntry);

	ELSE

		_kgArLogWrite.logLevel := arlogLEVEL_INFO;
		_kgArLogWrite.text := 'Create Ringbuffer: {##AttrVar1}';
		_kgArLogWrite.var1 := _kgRBcreateDFIIlog.wStatus;
		_kgArLogWrite.var2 := 0;
		_kgArLogWrite();

	END_IF

END_PROGRAM
```

#### hlDFIIExit.st - Exit code
```iecst
(********************************************************************
 * COPYRIGHT -- Microsoft
 ********************************************************************
 * Program: hlDFII
 * File: hlDFIIExit.st
 * Author: hunholz
 * Created: April 05, 2011
 * Changed: November 14, 2011
 ********************************************************************
 * Implementation of program hlDFII
 ********************************************************************)

PROGRAM _EXIT

	REPEAT
		_UdpClose(enable := TRUE, ident := _UdpOpen.ident);
		UNTIL
		_UdpClose.status <> ERR_FUB_BUSY
	END_REPEAT

	WHILE _eStep <> eSQLREQ_STEP_STOP DO

		CASE _eStep OF

			(* Beende Verbindungsaufbau, und baue dann die Verbindung wieder ab *)
			eSQLREQ_STEP_CONNECT_r:
				_DFII_Connect();
				IF _DFII_Connect.status <> ERR_FUB_BUSY THEN
					_eStep := eSQLREQ_STEP_DISCONNECT;
				END_IF

			(* Beende DFII_DBErrMsg *)
			eSQLREQ_STEP_GET_ERROR_r:
				_DFII_DBErrMsg();
				IF _DFII_DBErrMsg.status <> ERR_FUB_BUSY THEN
					_eStep := eSQLREQ_STEP_DISCONNECT;
				END_IF

			(* Beende Execute *)
			eSQLREQ_STEP_GPBC_r:
			eSQLREQ_STEP_WRMSG_r:
			eSQLREQ_STEP_WRCNTBATCHEVT_r:
			eSQLREQ_STEP_WRCNTCNTEVT_r:
			eSQLREQ_STEP_WRCNTTIMEVT_r:
			eSQLREQ_STEP_WRCNTDOSEVT_r:
			eSQLREQ_STEP_REGMACH_r:
				_DFII_DBExecute();
				IF _DFII_DBExecute.status <> ERR_FUB_BUSY THEN
					_eStep := eSQLREQ_STEP_DISCONNECT;
				END_IF

			(* Beende Fetch *)
			eSQLREQ_STEP_GPBC_FETCH_r:
				_DFII_DBFetch();
				IF _DFII_DBFetch.status <> ERR_FUB_BUSY THEN
					_eStep := eSQLREQ_STEP_DISCONNECT;
				END_IF

			(* Bende GetVal *)
			eSQLREQ_STEP_GPBC_GETVAL_r:
				_DFII_GetData();
				IF _DFII_GetData.status <> ERR_FUB_BUSY THEN
					_eStep := eSQLREQ_STEP_DISCONNECT;
				END_IF

			(* Baue Verbindung ab *)
			eSQLREQ_STEP_DISCONNECT:

				_DFII_Disconnect.enable := TRUE;
				_DFII_Disconnect.connectionIdent := _lConnectionIdent;
				_eStep := eSQLREQ_STEP_DISCONNECT_r;

			(* Warte bis Verbindung abgebaut ist *)
			eSQLREQ_STEP_DISCONNECT_r:

				_DFII_Disconnect();

				IF _DFII_Disconnect.status <> ERR_FUB_BUSY THEN
					_eStep := eSQLREQ_STEP_STOP;
				END_IF

			eSQLREQ_STEP_ERROR:

				_eStep := eSQLREQ_STEP_DISCONNECT;

			ELSE

				_eStep := eSQLREQ_STEP_DISCONNECT;

		END_CASE

	END_WHILE

END_PROGRAM
```

#### hlDFII.typ - Local data types
```iecst
(********************************************************************
 * COPYRIGHT -- Microsoft
 ********************************************************************
 * Program: hlDFII
 * File: hlDFII.typ
 * Author: hunholz
 * Created: April 05, 2011
 * Changed: Novemer 14, 2011
 ********************************************************************
 * Local data types of program hlDFII
 ********************************************************************)

TYPE
	SQLREQ_STEPS_enum :
		(
		eSQLREQ_STEP_STOP := 0,
		eSQLREQ_STEP_CONNECT := 10,
		eSQLREQ_STEP_CONNECT_r,
		eSQLREQ_STEP_DISCONNECT := 20,
		eSQLREQ_STEP_DISCONNECT_r,
		eSQLREQ_STEP_WAITFORCOMMAND := 30,
		eSQLREQ_STEP_GET_ERROR := 200,
		eSQLREQ_STEP_GET_ERROR_r,
		eSQLREQ_STEP_LOGRB_ERROR,
		eSQLREQ_STEP_LOG_ERROR,
		eSQLREQ_STEP_LOG_ERROR1,
		eSQLREQ_STEP_ERROR, (*Fehler Schritt*)
		eSQLREQ_STEP_DUMMY,
		eSQLREQ_STEP_GPBC := 40,
		eSQLREQ_STEP_GPBC_r,
		eSQLREQ_STEP_GPBC_FETCH,
		eSQLREQ_STEP_GPBC_FETCH_r,
		eSQLREQ_STEP_GPBC_GETVAL,
		eSQLREQ_STEP_GPBC_GETVAL_r,
		eSQLREQ_STEP_WRMSG := 50,
		eSQLREQ_STEP_WRMSG_r,
		eSQLREQ_STEP_WRCNTBATCHEVT := 60,
		eSQLREQ_STEP_WRCNTBATCHEVT_r,
		eSQLREQ_STEP_WRCNTCNTEVT := 70,
		eSQLREQ_STEP_WRCNTCNTEVT_r,
		eSQLREQ_STEP_WRCNTTIMEVT := 80,
		eSQLREQ_STEP_WRCNTTIMEVT_r,
		eSQLREQ_STEP_WRCNTDOSEVT := 90,
		eSQLREQ_STEP_WRCNTDOSEVT_r,
		eSQLREQ_STEP_REGMACH := 100,
		eSQLREQ_STEP_REGMACH_r,
		eSQLREQ_STEP_GETTIME := 110,
		eSQLREQ_STEP_GETTIME_r,
		eSQLREQ_STEP_GETTIME_FETCH,
		eSQLREQ_STEP_GETTIME_FETCH_r,
		eSQLREQ_STEP_GETTIME_GETVAL,
		eSQLREQ_STEP_GETTIME_GETVAL_r
		);
	cmdSqlReq_enum :
		(
		eCMD_SQLREQ_IDLE := 0, (*Nichts zu tun*)
		eCMD_SQLREQ_CONNECT := 10, (*Verbinde mit SQL-Server*)
		eCMD_SQLREQ_CONNECT_w, (*Warte auf Verbindung*)
		eCMD_SQLREQ_DISCONNECT := 20, (*Baue Verbindung zum SQL-Server wieder ab*)
		eCMD_SQLREQ_DISCONNECT_w, (*Warte bis Verbindung abgebaut ist*)
		eCMD_SQLREQ_GET_PROG_BY_CAT := 30, (*Lese Programmnumer*)
		eCMD_SQLREQ_GET_PROG_BY_CAT_w, (*Warte auf Programmnummer*)
		eCMD_SQLREQ_GET_LOAD_LIMIT := 40, (*Lese Beladegrenze*)
		eCMD_SQLREQ_GET_LOAD_LIMIT_w,
		eCMD_SQLREQ_SET_BATCHHEIGHT := 50, (*Schreibe Postenhöhe*)
		eCMD_SQLREQ_SET_BATCHHEIGHT_w,
		eCMD_SQLREQ_WRITE_MSG := 60, (*Meldungsevent und Zähler schreiben*)
		eCMD_SQLREQ_WRITE_MSG_w,
		eCMD_SQLREQ_WRITE_CNTBATCHEVT := 70,
		eCMD_SQLREQ_WRITE_CNTBATCHEVT_w,
		eCMD_SQLREQ_WRITE_CNTCNTEVT := 80,
		eCMD_SQLREQ_WRITE_CNTCNTEVT_w,
		eCMD_SQLREQ_WRITE_CNTTIMEVT := 90,
		eCMD_SQLREQ_WRITE_CNTTIMEVT_w,
		eCMD_SQLREQ_WRITE_CNTDOSEVT := 100,
		eCMD_SQLREQ_WRITE_CNTDOSEVT_W,
		eCMD_SQLREQ_WRITE_REGMACH := 110,
		eCMD_SQLREQ_WRITE_REGMACH_w,
		eCMD_SQLREQ_WRITE_GETTIME := 120,
		eCMD_SQLREQ_WRITE_GETTIME_w
		);
	_CacheEntry_typ : 	STRUCT
		dtTimeStamp : DATE_AND_TIME;
		sCategory : STRING[11];
		sProgShortName : STRING[15];
		bProgram : USINT;
	END_STRUCT;
END_TYPE
```

#### hlDFII.var - Local variables
```iecst
(********************************************************************
 * COPYRIGHT -- Microsoft
 ********************************************************************
 * Program: mnSqlReq
 * File: mnSqlReq.var
 * Author: hunholz
 * Created: April 05, 2011
 ********************************************************************
 * Local variables of program mnSqlReq
 ********************************************************************)
VAR
	_eStep : SQLREQ_STEPS_enum;
	_DFII_Connect : dbConnect;
	_lConnectionIdent : UDINT;
	_DFII_DBErrMsg : dbGetErrorMessage;
	_DFII_Disconnect : dbDisconnect;
	_sSQLstring : STRING[1023];
	_sMNo : STRING[15];
	_sCat : STRING[11];
	_DFII_DBExecute : dbExecuteSql;
	_DFII_DBFetch : dbFetchNextRow;
	_bCol : USINT;
	_DFII_GetData : dbGetData;
	_iProgNo : INT;
	_eCmdStep : cmdSqlReq_enum;
	_GTlastAction : DTGetTime;
	_GTCurrent : DTGetTime;
	_wCmdCnt : UINT := 0;
	_xReady : BOOL;
	_sOkt : STRING[5];
	_sDBserv : STRING[39];
	_bCntWrMsg : USINT;
	_sFunctionID : STRING[5];
	_sMsgNo : STRING[5];
	_sInstance : STRING[15];
	_sClass : STRING[3];
	_sEvent : STRING[5];
	_sTimeStamp : STRING[11];
	_sTime : STRING[11];
	_sValue : STRING[11];
	_bEventRegMach : USINT;
	_sShortName : STRING[15];
	TONrepReg : TON;
	_iFound : INT;
	_xInitDone : BOOL := FALSE;
END_VAR
VAR CONSTANT
	HLDFII_MSG_PROGBYCAT_ERR : UINT := 1000;
	HLDFII_MSG_MSGEVT_ERR : UINT := 1000;
	HLDFII_MSG_CNTBATCHEVT_ERR : UINT := 1000;
	HLDFII_MSG_CNTCNTEVT_ERR : UINT := 1000;
	HLDFII_MSG_CNTTIMEVT_ERR : UINT := 1000;
	HLDFII_MSG_CNTDOSEVT_ERR : UINT := 1000;
END_VAR
VAR
	_bCntWrCntBatchEvt : USINT;
	_bCntWrCntCntEvt : USINT;
	_kgUSINT16toGUID : kgUSINT16toGUID;
	_sUDINT : STRING[11];
	_kgGUIDtoSTRING : kgGUIDtoSTRING;
	_mnParam_datetimetoa : mnParam_datetimetoa;
	_ii : UINT;
	_xWaitReqMsgEvtIsZero : BOOL;
	_xWaitReqProgByCatIsZero : BOOL;
	_xWaitReqCntBatchIsZero : BOOL;
	_xWaitReqCntCntIsZero : BOOL;
	_xWaitReqCntTimIsZero : BOOL;
	_xWaitReqCntDosIsZero : BOOL;
	_bEventGetTime : USINT;
	_wHelpCmdCnt : UINT;
	TONrepGettime : TON;
	_diTime : DINT;
	_DTSetTime : DTSetTime;
	_kgArLogWrite : kgArLogWrite;
	_AsArLogCreate : AsArLogCreate;
	_AsArLogGetInfo : AsArLogGetInfo;
END_VAR
VAR RETAIN
	_wPtrRBwrite : UINT;
	_wPtrRBread : UINT;
	_wPtrRBloc : UINT;
END_VAR
VAR
	_xRBReady : BOOL;
	_InsertRB : kgRBinsert;
	_ReadRB : kgRBread;
	_UdpOpen : UdpOpen;
	_wStepUdp : UINT;
	_sLogEntry : STRING[511];
	_UdpSend : UdpSend;
	_sUdpHost : STRING[15];
	_UdpClose : UdpClose;
	_sAction : STRING[31];
	_sPkgName : STRING[11];
	_VerStruc : MoVerStruc_typ;
	_sMark : STRING[31];
	_bCntWrCntTimeEvt : USINT;
	_bCntWrCntDoseEvt : USINT;
	_sDoseName : STRING[23];
END_VAR
VAR RETAIN
	_wPtrRBstart : UINT;
END_VAR
VAR
	_kgRBcreateDFIIlog : kgRBcreate;
	_sLogEntryI : STRING[511];
	_wStartDebug : UINT;
	_sDebugSQLstring : REFERENCE TO STRING[31];
	_sSQLBatchEventString : STRING[1023];
	_idxCustomer : UINT;
	_rLoadfactor : REAL;
	_diColIdxFor : DINT;
	_diColIdxBack : DINT;
	_sName : STRING[31];
END_VAR
```

### hlDFII_History.txt
```
1.03.0		28.9.2011	AH Auf mnParam 0.05.0 umgestellt
1.04.0		11.10.2011	AH Auf mnParam 0.06.0 umgestellt, Maschinennummer kommt aus Datei
1.04.1		18.11.2011	AH Zwischenversion. Maschinenregistrierung startet jetzt automatisch.
						AH Attribute werden mit in die Meldungshistorie eingetragen
1.05.0		03.11.2011	AH Umstellung auf AS 3.0.90. IF ist eindeutig mit Ein- und Ausgangskanal definiert
			14.11.2011	AH Schnittstelle zu mnCnt umgestellt
1.06.0		21.12.2011	AH SPS-Log und UDP-Logging eingeführt
						AH Fehlerhandling geändert. Bei Fehlern wird grundsätzlich die Verbindung abgebaut.
1.07.0		03.01.2012	AH Packetversion wird in hlDFIIStatAd ausgegeben
1.08.0		12.01.2012	AH Kategorie-Programm-Zuordnung wird gecachet
1.09.0		24.01.2012	AH Anpassung an KGStandard 1.13.0 (Ringbuffer)
1.10.0		26.01.2012  AH Erweiterter Substatus für Zeitzähler mnCnt 0.14.0
1.10.1		07.02.2012  AH Schließendes Anführungszeichen im SQL-String Batch-Event für die MachineID fehlte
						AH Logeintrag erweitert
1.10.2		07.02.2012	AH Bei Batchevent mit 0 Teilposten hat sich die Sendeschrittkette aufgehängt
1.10.3		07.02.2012	AH GO ist kein gültiger TSQL-Befehl
1.10.4		07.02.2012	AH SQL-String Batchevent zu Debugzwecken kopiert. Log-String auf 511 Zeichen verlängert.
1.10.5		09.02.2012	AH Ziel- und Quellnamen für Postenevent ergänzt.
1.10.6		10.02.2012	AH Bei spInsEventStatItem_StateTime ein Komma zu viel
1.11.0		10.02.2012	AH Batchevent gibt jetzt immer Quell- und Zielort an. Dazu ist auch mnCnt 0.15.0 notwendig
1.11.1		10.02.2012	AH Wieder ein Komma zu viel
1.11.2		10.02.2012	AH Anführungszeichen hinter Maschinennummer oftmals zu wenig
1.11.3		10.02.2012	AH FromOutside und ToOutside müssen beim BatchEvent immer beide definiert sein
1.12.0		13.02.2012	AH Einige Korrekturen auf Anregung von Thomas Horn (Fehler in Strings, Komma usw.)
						   Anpassung an mnCnt 0.16.0
1.12.1		14.02.2012	AH Error-Logging erweitert und Debugging korrigiert. Logging-Port ist jetzt per Konstante definiert
						   HLDFII_UDP_PORT_LOG4NET
1.12.2		14.02.2012	AH Jetzt sollte auch der richtige String an Log4Net geschickt werden
1.13.0		20.02.2012	AH Client muss per Konfiguration freigeschaltet werden und kann per Parameter deaktiviert werden
							- Package gibt im IFhlDFII.Out.wStatus den aktuellen Status OK, Init oder Disabled aus (siehe Konstanten)
1.14.0		13.03.2012	AH Client muss per Konstante freigeschaltet werden. Andernfalls läuft er nicht an. Parameter von 1.13.0 entfallen wieder.
						   Mehr UDP-Logging
1.14.1		20.03.2012	AH Abhängigkeiten
1.14.2		28.03.2012	AH Bugfix: Logger. Parameter Start wurde nicht übergeben.
						   Connectionstring: Entweder Port oder Instanz.
1.15.0		03.04.2012	AH Category Cache entfernt.
						   xConnected eingeführt
1.16.0		11.04.2012	AH Maschinenregistrierung sendet jetzt auch den Maschinennamen
```

### Package Logical/Mewa/KGFramework/Pkg_hlKanLink - Kanlink 

### hlKanLink.var - Global variables
```iecst
(********************************************************************
 * COPYRIGHT -- Bernecker + Rainer
 ********************************************************************
 * File: Global.var
 * Author: Bernecker + Rainer
 * Created: June 02, 2008
 ********************************************************************
 * Global variables of project LibAsUDP
 ********************************************************************)
VAR
	hlKanLinkStatAd : hlKanLinkStatAd_typ;
	hlKanLinkStat : Stat_typ;
	IFhlKanLink : IFhlKanLink_Typ;
END_VAR
(*Konstanten*)
VAR CONSTANT
	HLKANLINK_MSG_NO_STRUCDEF : UINT := 60000;
END_VAR
```

### Program Logical/Mewa/KGFramework/Pkg_hlKanLink/hlKanLink (IEC, version 0.90.0) - A new program
